LIN {X -6.617,Y -42.351,Z -210.966,A -90.000,B 90.000,C 0.000} C_DIS
LIN {X -6.280,Y -42.371,Z -210.884,A -90.000,B 90.000,C 0.000} C_DIS
LIN {X -6.014,Y -42.388,Z -210.830,A -90.000,B 90.000,C 0.000} C_DIS
LIN {X -5.294,Y -42.439,Z -210.703,A -90.000,B 90.000,C 0.000} C_DIS
LIN {X -5.055,Y -42.457,Z -210.668,A -90.000,B 90.000,C 0.000} C_DIS
LIN {X -4.913,Y -42.469,Z -210.653,A -90.000,B 90.000,C 0.000} C_DIS
LIN {X -4.678,Y -42.489,Z -210.636,A -90.000,B 90.000,C 0.000} C_DIS
LIN {X -4.349,Y -42.521,Z -210.624,A -90.000,B 90.000,C 0.000} C_DIS
LIN {X -4.051,Y -42.551,Z -210.626,A -90.000,B 90.000,C 0.000} C_DIS
LIN {X -3.773,Y -42.581,Z -210.638,A -90.000,B 90.000,C 0.000} C_DIS
LIN {X -3.082,Y -42.611,Z -210.410,A -90.000,B 90.000,C 0.000} C_DIS
LIN {X -2.709,Y -42.612,Z -210.205,A -90.000,B 90.000,C 0.000} C_DIS
LIN {X -2.509,Y -42.614,Z -210.106,A -90.000,B 90.000,C 0.000} C_DIS
LIN {X -2.183,Y -42.620,Z -209.957,A -90.000,B 90.000,C 0.000} C_DIS
LIN {X -2.016,Y -42.624,Z -209.889,A -90.000,B 90.000,C 0.000} C_DIS
LIN {X -1.766,Y -42.632,Z -209.800,A -90.000,B 90.000,C 0.000} C_DIS
LIN {X -1.327,Y -42.645,Z -209.666,A -90.000,B 90.000,C 0.000} C_DIS
LIN {X -1.055,Y -42.655,Z -209.597,A -90.000,B 90.000,C 0.000} C_DIS
LIN {X -0.921,Y -42.661,Z -209.569,A -90.000,B 90.000,C 0.000} C_DIS
LIN {X -0.790,Y -42.670,Z -209.542,A -90.000,B 90.000,C 0.000} C_DIS
LIN {X -0.184,Y -42.653,Z -208.934,A -90.000,B 90.000,C 0.000} C_DIS
LIN {X -0.036,Y -42.650,Z -208.795,A -90.000,B 90.000,C 0.000} C_DIS
LIN {X 0.358,Y -42.637,Z -208.433,A -90.000,B 90.000,C 0.000} C_DIS
LIN {X 2.070,Y -42.427,Z -205.938,A -90.000,B 90.000,C 0.000} C_DIS
LIN {X 2.234,Y -42.419,Z -205.708,A -90.000,B 90.000,C 0.000} C_DIS
LIN {X 2.733,Y -42.394,Z -205.030,A -90.000,B 90.000,C 0.000} C_DIS
LIN {X 3.270,Y -42.350,Z -204.307,A -90.000,B 90.000,C 0.000} C_DIS
LIN {X 4.497,Y -42.165,Z -202.176,A -90.000,B 90.000,C 0.000} C_DIS
LIN {X 4.596,Y -42.148,Z -202.016,A -90.000,B 90.000,C 0.000} C_DIS
LIN {X 6.267,Y -41.968,Z -199.269,A -90.000,B 90.000,C 0.000} C_DIS
LIN {X 6.453,Y -41.942,Z -198.966,A -90.000,B 90.000,C 0.000} C_DIS
LIN {X 6.699,Y -41.891,Z -198.498,A -90.000,B 90.000,C 0.000} C_DIS
LIN {X 7.020,Y -41.828,Z -197.909,A -90.000,B 90.000,C 0.000} C_DIS
LIN {X 7.766,Y -41.714,Z -196.530,A -90.000,B 90.000,C 0.000} C_DIS
LIN {X 7.949,Y -41.691,Z -196.212,A -90.000,B 90.000,C 0.000} C_DIS
LIN {X 9.284,Y -41.563,Z -193.973,A -90.000,B 90.000,C 0.000} C_DIS
LIN {X 9.444,Y -41.549,Z -193.721,A -90.000,B 90.000,C 0.000} C_DIS
LIN {X 9.586,Y -41.533,Z -193.478,A -90.000,B 90.000,C 0.000} C_DIS
LIN {X 10.446,Y -41.437,Z -192.021,A -90.000,B 90.000,C 0.000} C_DIS
LIN {X 10.972,Y -41.378,Z -191.131,A -90.000,B 90.000,C 0.000} C_DIS
LIN {X 11.489,Y -41.308,Z -190.267,A -90.000,B 90.000,C 0.000} C_DIS
LIN {X 11.489,Y -60.000,Z -190.267,A -90.000,B 90.000,C 0.000} C_DIS
LIN {X -12.262,Y -60.000,Z -210.299,A -90.000,B 90.000,C 0.000} C_DIS
LIN {X -12.262,Y -41.308,Z -210.299,A -90.000,B 90.000,C 0.000} C_DIS
LIN {X -11.900,Y -41.347,Z -210.184,A -90.000,B 90.000,C 0.000} C_DIS
LIN {X -11.506,Y -41.394,Z -210.074,A -90.000,B 90.000,C 0.000} C_DIS
LIN {X -11.190,Y -41.436,Z -210.001,A -90.000,B 90.000,C 0.000} C_DIS
LIN {X -11.051,Y -41.456,Z -209.972,A -90.000,B 90.000,C 0.000} C_DIS
LIN {X -10.725,Y -41.505,Z -209.911,A -90.000,B 90.000,C 0.000} C_DIS
LIN {X -10.408,Y -41.557,Z -209.864,A -90.000,B 90.000,C 0.000} C_DIS
LIN {X -9.634,Y -41.647,Z -209.785,A -90.000,B 90.000,C 0.000} C_DIS
LIN {X -9.462,Y -41.666,Z -209.768,A -90.000,B 90.000,C 0.000} C_DIS
LIN {X -9.236,Y -41.684,Z -209.720,A -90.000,B 90.000,C 0.000} C_DIS
LIN {X -8.688,Y -41.735,Z -209.603,A -90.000,B 90.000,C 0.000} C_DIS
LIN {X -8.324,Y -41.772,Z -209.525,A -90.000,B 90.000,C 0.000} C_DIS
LIN {X -8.206,Y -41.777,Z -209.473,A -90.000,B 90.000,C 0.000} C_DIS
LIN {X -8.132,Y -41.782,Z -209.447,A -90.000,B 90.000,C 0.000} C_DIS
LIN {X -7.916,Y -41.793,Z -209.356,A -90.000,B 90.000,C 0.000} C_DIS
LIN {X -7.715,Y -41.806,Z -209.283,A -90.000,B 90.000,C 0.000} C_DIS
LIN {X -7.389,Y -41.830,Z -209.175,A -90.000,B 90.000,C 0.000} C_DIS
LIN {X -7.217,Y -41.843,Z -209.124,A -90.000,B 90.000,C 0.000} C_DIS
LIN {X -7.050,Y -41.858,Z -209.077,A -90.000,B 90.000,C 0.000} C_DIS
LIN {X -6.640,Y -41.895,Z -208.975,A -90.000,B 90.000,C 0.000} C_DIS
LIN {X -6.321,Y -41.928,Z -208.907,A -90.000,B 90.000,C 0.000} C_DIS
LIN {X -5.544,Y -42.012,Z -208.765,A -90.000,B 90.000,C 0.000} C_DIS
LIN {X -5.228,Y -42.049,Z -208.717,A -90.000,B 90.000,C 0.000} C_DIS
LIN {X -5.016,Y -42.076,Z -208.694,A -90.000,B 90.000,C 0.000} C_DIS
LIN {X -4.805,Y -42.103,Z -208.678,A -90.000,B 90.000,C 0.000} C_DIS
LIN {X -4.663,Y -42.117,Z -208.671,A -90.000,B 90.000,C 0.000} C_DIS
LIN {X -4.355,Y -42.149,Z -208.659,A -90.000,B 90.000,C 0.000} C_DIS
LIN {X -4.025,Y -42.185,Z -208.660,A -90.000,B 90.000,C 0.000} C_DIS
LIN {X -3.857,Y -42.193,Z -208.605,A -90.000,B 90.000,C 0.000} C_DIS
LIN {X -3.580,Y -42.193,Z -208.454,A -90.000,B 90.000,C 0.000} C_DIS
LIN {X -3.315,Y -42.196,Z -208.323,A -90.000,B 90.000,C 0.000} C_DIS
LIN {X -2.989,Y -42.202,Z -208.174,A -90.000,B 90.000,C 0.000} C_DIS
LIN {X -2.844,Y -42.206,Z -208.114,A -90.000,B 90.000,C 0.000} C_DIS
LIN {X -2.716,Y -42.210,Z -208.062,A -90.000,B 90.000,C 0.000} C_DIS
LIN {X -2.412,Y -42.229,Z -207.951,A -90.000,B 90.000,C 0.000} C_DIS
LIN {X -2.184,Y -42.245,Z -207.877,A -90.000,B 90.000,C 0.000} C_DIS
LIN {X -1.891,Y -42.266,Z -207.785,A -90.000,B 90.000,C 0.000} C_DIS
LIN {X -1.797,Y -42.273,Z -207.758,A -90.000,B 90.000,C 0.000} C_DIS
LIN {X -1.778,Y -42.274,Z -207.753,A -90.000,B 90.000,C 0.000} C_DIS
LIN {X -1.529,Y -42.262,Z -207.506,A -90.000,B 90.000,C 0.000} C_DIS
LIN {X -1.146,Y -42.248,Z -207.152,A -90.000,B 90.000,C 0.000} C_DIS
LIN {X -0.566,Y -42.173,Z -206.308,A -90.000,B 90.000,C 0.000} C_DIS
LIN {X 0.472,Y -42.006,Z -204.812,A -90.000,B 90.000,C 0.000} C_DIS
LIN {X 0.654,Y -41.989,Z -204.560,A -90.000,B 90.000,C 0.000} C_DIS
LIN {X 1.498,Y -41.917,Z -203.424,A -90.000,B 90.000,C 0.000} C_DIS
LIN {X 1.621,Y -41.903,Z -203.259,A -90.000,B 90.000,C 0.000} C_DIS
LIN {X 2.825,Y -41.665,Z -201.198,A -90.000,B 90.000,C 0.000} C_DIS
LIN {X 2.924,Y -41.649,Z -201.038,A -90.000,B 90.000,C 0.000} C_DIS
LIN {X 3.144,Y -41.624,Z -200.676,A -90.000,B 90.000,C 0.000} C_DIS
LIN {X 3.568,Y -41.563,Z -199.988,A -90.000,B 90.000,C 0.000} C_DIS
LIN {X 4.759,Y -41.384,Z -198.058,A -90.000,B 90.000,C 0.000} C_DIS
LIN {X 4.988,Y -41.334,Z -197.625,A -90.000,B 90.000,C 0.000} C_DIS
LIN {X 5.113,Y -41.308,Z -197.396,A -90.000,B 90.000,C 0.000} C_DIS
LIN {X 5.113,Y -60.000,Z -197.396,A -90.000,B 90.000,C 0.000} C_DIS
LIN {X -7.484,Y -60.000,Z -207.204,A -90.000,B 90.000,C 0.000} C_DIS
LIN {X -7.484,Y -41.308,Z -207.204,A -90.000,B 90.000,C 0.000} C_DIS
LIN {X -6.986,Y -41.355,Z -207.081,A -90.000,B 90.000,C 0.000} C_DIS
LIN {X -6.613,Y -41.394,Z -207.002,A -90.000,B 90.000,C 0.000} C_DIS
LIN {X -5.770,Y -41.488,Z -206.848,A -90.000,B 90.000,C 0.000} C_DIS
LIN {X -5.453,Y -41.526,Z -206.800,A -90.000,B 90.000,C 0.000} C_DIS
LIN {X -5.161,Y -41.564,Z -206.766,A -90.000,B 90.000,C 0.000} C_DIS
LIN {X -4.857,Y -41.606,Z -206.741,A -90.000,B 90.000,C 0.000} C_DIS
LIN {X -4.638,Y -41.638,Z -206.729,A -90.000,B 90.000,C 0.000} C_DIS
LIN {X -4.424,Y -41.670,Z -206.718,A -90.000,B 90.000,C 0.000} C_DIS
LIN {X -4.164,Y -41.683,Z -206.587,A -90.000,B 90.000,C 0.000} C_DIS
LIN {X -3.727,Y -41.709,Z -206.382,A -90.000,B 90.000,C 0.000} C_DIS
LIN {X -3.429,Y -41.730,Z -206.256,A -90.000,B 90.000,C 0.000} C_DIS
LIN {X -3.096,Y -41.758,Z -206.131,A -90.000,B 90.000,C 0.000} C_DIS
LIN {X -2.982,Y -41.767,Z -206.090,A -90.000,B 90.000,C 0.000} C_DIS
LIN {X -2.792,Y -41.785,Z -206.027,A -90.000,B 90.000,C 0.000} C_DIS
LIN {X -2.642,Y -41.778,Z -205.889,A -90.000,B 90.000,C 0.000} C_DIS
LIN {X -1.365,Y -41.555,Z -204.057,A -90.000,B 90.000,C 0.000} C_DIS
LIN {X -1.115,Y -41.506,Z -203.702,A -90.000,B 90.000,C 0.000} C_DIS
LIN {X -1.083,Y -41.500,Z -203.658,A -90.000,B 90.000,C 0.000} C_DIS
LIN {X -0.913,Y -41.478,Z -203.427,A -90.000,B 90.000,C 0.000} C_DIS
LIN {X -0.012,Y -41.369,Z -202.229,A -90.000,B 90.000,C 0.000} C_DIS
LIN {X 0.278,Y -41.308,Z -201.734,A -90.000,B 90.000,C 0.000} C_DIS
LIN {X 0.278,Y -60.000,Z -201.734,A -90.000,B 90.000,C 0.000} C_DIS
LIN {X -23.050,Y -60.000,Z -133.482,A -90.000,B 90.000,C 0.000} C_DIS
LIN {X -23.050,Y -41.308,Z -133.482,A -90.000,B 90.000,C 0.000} C_DIS
LIN {X -23.070,Y -41.317,Z -133.385,A -90.000,B 90.000,C 0.000} C_DIS
LIN {X -23.094,Y -41.329,Z -133.252,A -90.000,B 90.000,C 0.000} C_DIS
LIN {X -23.314,Y -41.439,Z -131.911,A -90.000,B 90.000,C 0.000} C_DIS
LIN {X -23.329,Y -41.449,Z -131.802,A -90.000,B 90.000,C 0.000} C_DIS
LIN {X -23.404,Y -41.504,Z -131.165,A -90.000,B 90.000,C 0.000} C_DIS
LIN {X -23.458,Y -41.576,Z -130.456,A -90.000,B 90.000,C 0.000} C_DIS
LIN {X -23.470,Y -41.599,Z -130.246,A -90.000,B 90.000,C 0.000} C_DIS
LIN {X -23.473,Y -41.621,Z -130.071,A -90.000,B 90.000,C 0.000} C_DIS
LIN {X -23.473,Y -41.634,Z -129.976,A -90.000,B 90.000,C 0.000} C_DIS
LIN {X -23.470,Y -41.652,Z -129.815,A -90.000,B 90.000,C 0.000} C_DIS
LIN {X -23.462,Y -41.671,Z -129.600,A -90.000,B 90.000,C 0.000} C_DIS
LIN {X -23.484,Y -41.694,Z -129.239,A -90.000,B 90.000,C 0.000} C_DIS
LIN {X -23.533,Y -41.742,Z -128.346,A -90.000,B 90.000,C 0.000} C_DIS
LIN {X -23.555,Y -41.785,Z -127.639,A -90.000,B 90.000,C 0.000} C_DIS
LIN {X -23.575,Y -41.830,Z -127.087,A -90.000,B 90.000,C 0.000} C_DIS
LIN {X -23.574,Y -41.836,Z -127.029,A -90.000,B 90.000,C 0.000} C_DIS
LIN {X -23.576,Y -41.850,Z -126.858,A -90.000,B 90.000,C 0.000} C_DIS
LIN {X -23.569,Y -41.874,Z -126.625,A -90.000,B 90.000,C 0.000} C_DIS
LIN {X -23.533,Y -41.955,Z -125.844,A -90.000,B 90.000,C 0.000} C_DIS
LIN {X -23.511,Y -41.992,Z -125.277,A -90.000,B 90.000,C 0.000} C_DIS
LIN {X -23.515,Y -41.993,Z -125.243,A -90.000,B 90.000,C 0.000} C_DIS
LIN {X -23.643,Y -42.000,Z -124.602,A -90.000,B 90.000,C 0.000} C_DIS
LIN {X -23.792,Y -42.013,Z -123.757,A -90.000,B 90.000,C 0.000} C_DIS
LIN {X -24.070,Y -42.088,Z -122.244,A -90.000,B 90.000,C 0.000} C_DIS
LIN {X -24.088,Y -42.092,Z -122.140,A -90.000,B 90.000,C 0.000} C_DIS
LIN {X -24.107,Y -42.093,Z -122.030,A -90.000,B 90.000,C 0.000} C_DIS
LIN {X -24.170,Y -42.098,Z -121.672,A -90.000,B 90.000,C 0.000} C_DIS
LIN {X -24.188,Y -42.102,Z -121.571,A -90.000,B 90.000,C 0.000} C_DIS
LIN {X -24.313,Y -42.107,Z -121.167,A -90.000,B 90.000,C 0.000} C_DIS
LIN {X -24.362,Y -42.107,Z -121.018,A -90.000,B 90.000,C 0.000} C_DIS
LIN {X -24.809,Y -42.092,Z -119.638,A -90.000,B 90.000,C 0.000} C_DIS
LIN {X -25.186,Y -42.121,Z -118.503,A -90.000,B 90.000,C 0.000} C_DIS
LIN {X -25.572,Y -42.137,Z -117.266,A -90.000,B 90.000,C 0.000} C_DIS
LIN {X -25.886,Y -42.145,Z -116.322,A -90.000,B 90.000,C 0.000} C_DIS
LIN {X -25.961,Y -42.146,Z -116.092,A -90.000,B 90.000,C 0.000} C_DIS
LIN {X -26.400,Y -42.139,Z -114.737,A -90.000,B 90.000,C 0.000} C_DIS
LIN {X -26.782,Y -42.128,Z -113.563,A -90.000,B 90.000,C 0.000} C_DIS
LIN {X -27.447,Y -42.107,Z -111.546,A -90.000,B 90.000,C 0.000} C_DIS
LIN {X -27.639,Y -42.097,Z -110.961,A -90.000,B 90.000,C 0.000} C_DIS
LIN {X -27.709,Y -42.085,Z -110.741,A -90.000,B 90.000,C 0.000} C_DIS
LIN {X -27.755,Y -42.074,Z -110.581,A -90.000,B 90.000,C 0.000} C_DIS
LIN {X -27.902,Y -42.042,Z -110.029,A -90.000,B 90.000,C 0.000} C_DIS
LIN {X -27.980,Y -42.025,Z -109.706,A -90.000,B 90.000,C 0.000} C_DIS
LIN {X -28.117,Y -41.997,Z -109.053,A -90.000,B 90.000,C 0.000} C_DIS
LIN {X -28.358,Y -41.959,Z -107.920,A -90.000,B 90.000,C 0.000} C_DIS
LIN {X -28.564,Y -41.915,Z -106.996,A -90.000,B 90.000,C 0.000} C_DIS
LIN {X -28.601,Y -41.908,Z -106.827,A -90.000,B 90.000,C 0.000} C_DIS
LIN {X -28.724,Y -41.886,Z -106.164,A -90.000,B 90.000,C 0.000} C_DIS
LIN {X -28.845,Y -41.853,Z -105.495,A -90.000,B 90.000,C 0.000} C_DIS
LIN {X -28.878,Y -41.839,Z -105.307,A -90.000,B 90.000,C 0.000} C_DIS
LIN {X -29.130,Y -41.699,Z -103.813,A -90.000,B 90.000,C 0.000} C_DIS
LIN {X -29.182,Y -41.668,Z -103.454,A -90.000,B 90.000,C 0.000} C_DIS
LIN {X -29.224,Y -41.644,Z -103.086,A -90.000,B 90.000,C 0.000} C_DIS
LIN {X -29.270,Y -41.615,Z -102.509,A -90.000,B 90.000,C 0.000} C_DIS
LIN {X -29.284,Y -41.604,Z -102.259,A -90.000,B 90.000,C 0.000} C_DIS
LIN {X -29.288,Y -41.597,Z -101.997,A -90.000,B 90.000,C 0.000} C_DIS
LIN {X -29.280,Y -41.590,Z -101.741,A -90.000,B 90.000,C 0.000} C_DIS
LIN {X -29.250,Y -41.584,Z -101.188,A -90.000,B 90.000,C 0.000} C_DIS
LIN {X -29.178,Y -41.548,Z -100.027,A -90.000,B 90.000,C 0.000} C_DIS
LIN {X -29.153,Y -41.527,Z -99.698,A -90.000,B 90.000,C 0.000} C_DIS
LIN {X -29.138,Y -41.516,Z -99.489,A -90.000,B 90.000,C 0.000} C_DIS
LIN {X -29.120,Y -41.500,Z -99.279,A -90.000,B 90.000,C 0.000} C_DIS
LIN {X -29.077,Y -41.476,Z -98.905,A -90.000,B 90.000,C 0.000} C_DIS
LIN {X -29.047,Y -41.466,Z -98.703,A -90.000,B 90.000,C 0.000} C_DIS
LIN {X -29.015,Y -41.459,Z -98.520,A -90.000,B 90.000,C 0.000} C_DIS
LIN {X -28.923,Y -41.447,Z -98.052,A -90.000,B 90.000,C 0.000} C_DIS
LIN {X -28.723,Y -41.430,Z -96.999,A -90.000,B 90.000,C 0.000} C_DIS
LIN {X -28.657,Y -41.423,Z -96.681,A -90.000,B 90.000,C 0.000} C_DIS
LIN {X -28.528,Y -41.392,Z -96.095,A -90.000,B 90.000,C 0.000} C_DIS
LIN {X -28.491,Y -41.386,Z -95.924,A -90.000,B 90.000,C 0.000} C_DIS
LIN {X -28.434,Y -41.380,Z -95.697,A -90.000,B 90.000,C 0.000} C_DIS
LIN {X -28.370,Y -41.376,Z -95.462,A -90.000,B 90.000,C 0.000} C_DIS
LIN {X -28.232,Y -41.376,Z -95.022,A -90.000,B 90.000,C 0.000} C_DIS
LIN {X -28.161,Y -41.380,Z -94.821,A -90.000,B 90.000,C 0.000} C_DIS
LIN {X -27.995,Y -41.393,Z -94.384,A -90.000,B 90.000,C 0.000} C_DIS
LIN {X -27.971,Y -41.392,Z -94.325,A -90.000,B 90.000,C 0.000} C_DIS
LIN {X -27.835,Y -41.387,Z -93.984,A -90.000,B 90.000,C 0.000} C_DIS
LIN {X -27.746,Y -41.381,Z -93.769,A -90.000,B 90.000,C 0.000} C_DIS
LIN {X -27.107,Y -41.358,Z -92.328,A -90.000,B 90.000,C 0.000} C_DIS
LIN {X -26.960,Y -41.359,Z -92.025,A -90.000,B 90.000,C 0.000} C_DIS
LIN {X -26.939,Y -41.360,Z -91.984,A -90.000,B 90.000,C 0.000} C_DIS
LIN {X -26.749,Y -41.354,Z -91.643,A -90.000,B 90.000,C 0.000} C_DIS
LIN {X -26.597,Y -41.354,Z -91.391,A -90.000,B 90.000,C 0.000} C_DIS
LIN {X -26.044,Y -41.374,Z -90.536,A -90.000,B 90.000,C 0.000} C_DIS
LIN {X -25.785,Y -41.388,Z -90.154,A -90.000,B 90.000,C 0.000} C_DIS
LIN {X -25.678,Y -41.396,Z -89.994,A -90.000,B 90.000,C 0.000} C_DIS
LIN {X -25.507,Y -41.402,Z -89.745,A -90.000,B 90.000,C 0.000} C_DIS
LIN {X -25.112,Y -41.397,Z -89.178,A -90.000,B 90.000,C 0.000} C_DIS
LIN {X -24.983,Y -41.397,Z -89.006,A -90.000,B 90.000,C 0.000} C_DIS
LIN {X -24.826,Y -41.399,Z -88.802,A -90.000,B 90.000,C 0.000} C_DIS
LIN {X -24.722,Y -41.402,Z -88.675,A -90.000,B 90.000,C 0.000} C_DIS
LIN {X -24.486,Y -41.412,Z -88.401,A -90.000,B 90.000,C 0.000} C_DIS
LIN {X -23.946,Y -41.445,Z -87.813,A -90.000,B 90.000,C 0.000} C_DIS
LIN {X -23.608,Y -41.453,Z -87.454,A -90.000,B 90.000,C 0.000} C_DIS
LIN {X -22.465,Y -41.470,Z -86.254,A -90.000,B 90.000,C 0.000} C_DIS
LIN {X -22.294,Y -41.476,Z -86.088,A -90.000,B 90.000,C 0.000} C_DIS
LIN {X -22.148,Y -41.484,Z -85.957,A -90.000,B 90.000,C 0.000} C_DIS
LIN {X -21.990,Y -41.494,Z -85.821,A -90.000,B 90.000,C 0.000} C_DIS
LIN {X -21.611,Y -41.517,Z -85.511,A -90.000,B 90.000,C 0.000} C_DIS
LIN {X -21.025,Y -41.548,Z -85.034,A -90.000,B 90.000,C 0.000} C_DIS
LIN {X -20.092,Y -41.578,Z -84.281,A -90.000,B 90.000,C 0.000} C_DIS
LIN {X -19.821,Y -41.583,Z -84.065,A -90.000,B 90.000,C 0.000} C_DIS
LIN {X -19.531,Y -41.587,Z -83.835,A -90.000,B 90.000,C 0.000} C_DIS
LIN {X -19.253,Y -41.588,Z -83.630,A -90.000,B 90.000,C 0.000} C_DIS
LIN {X -19.000,Y -41.592,Z -83.456,A -90.000,B 90.000,C 0.000} C_DIS
LIN {X -18.820,Y -41.594,Z -83.345,A -90.000,B 90.000,C 0.000} C_DIS
LIN {X -18.604,Y -41.598,Z -83.216,A -90.000,B 90.000,C 0.000} C_DIS
LIN {X -18.307,Y -41.608,Z -83.053,A -90.000,B 90.000,C 0.000} C_DIS
LIN {X -17.615,Y -41.631,Z -82.678,A -90.000,B 90.000,C 0.000} C_DIS
LIN {X -16.357,Y -41.640,Z -82.007,A -90.000,B 90.000,C 0.000} C_DIS
LIN {X -16.157,Y -41.644,Z -81.909,A -90.000,B 90.000,C 0.000} C_DIS
LIN {X -15.796,Y -41.652,Z -81.743,A -90.000,B 90.000,C 0.000} C_DIS
LIN {X -15.527,Y -41.656,Z -81.627,A -90.000,B 90.000,C 0.000} C_DIS
LIN {X -15.356,Y -41.651,Z -81.555,A -90.000,B 90.000,C 0.000} C_DIS
LIN {X -14.632,Y -41.625,Z -81.254,A -90.000,B 90.000,C 0.000} C_DIS
LIN {X -14.380,Y -41.619,Z -81.159,A -90.000,B 90.000,C 0.000} C_DIS
LIN {X -14.313,Y -41.617,Z -81.134,A -90.000,B 90.000,C 0.000} C_DIS
LIN {X -13.263,Y -41.602,Z -80.775,A -90.000,B 90.000,C 0.000} C_DIS
LIN {X -13.022,Y -41.593,Z -80.697,A -90.000,B 90.000,C 0.000} C_DIS
LIN {X -12.835,Y -41.588,Z -80.644,A -90.000,B 90.000,C 0.000} C_DIS
LIN {X -12.618,Y -41.584,Z -80.588,A -90.000,B 90.000,C 0.000} C_DIS
LIN {X -11.074,Y -41.571,Z -80.238,A -90.000,B 90.000,C 0.000} C_DIS
LIN {X -10.804,Y -41.562,Z -80.179,A -90.000,B 90.000,C 0.000} C_DIS
LIN {X -9.749,Y -41.484,Z -79.972,A -90.000,B 90.000,C 0.000} C_DIS
LIN {X -9.567,Y -41.473,Z -79.943,A -90.000,B 90.000,C 0.000} C_DIS
LIN {X -9.291,Y -41.458,Z -79.904,A -90.000,B 90.000,C 0.000} C_DIS
LIN {X -8.345,Y -41.422,Z -79.809,A -90.000,B 90.000,C 0.000} C_DIS
LIN {X -8.092,Y -41.407,Z -79.786,A -90.000,B 90.000,C 0.000} C_DIS
LIN {X -6.966,Y -41.348,Z -79.697,A -90.000,B 90.000,C 0.000} C_DIS
LIN {X -6.019,Y -41.308,Z -79.651,A -90.000,B 90.000,C 0.000} C_DIS
LIN {X -6.019,Y -60.000,Z -79.651,A -90.000,B 90.000,C 0.000} C_DIS
LIN {X 25.151,Y -60.000,Z -82.979,A -90.000,B 90.000,C 0.000} C_DIS
LIN {X 25.151,Y -41.308,Z -82.979,A -90.000,B 90.000,C 0.000} C_DIS
LIN {X 25.401,Y -41.345,Z -82.958,A -90.000,B 90.000,C 0.000} C_DIS
LIN {X 26.505,Y -41.507,Z -82.878,A -90.000,B 90.000,C 0.000} C_DIS
LIN {X 27.673,Y -41.657,Z -82.800,A -90.000,B 90.000,C 0.000} C_DIS
LIN {X 27.698,Y -41.660,Z -82.799,A -90.000,B 90.000,C 0.000} C_DIS
LIN {X 28.017,Y -41.696,Z -82.752,A -90.000,B 90.000,C 0.000} C_DIS
LIN {X 28.158,Y -41.713,Z -82.736,A -90.000,B 90.000,C 0.000} C_DIS
LIN {X 28.252,Y -41.725,Z -82.727,A -90.000,B 90.000,C 0.000} C_DIS
LIN {X 28.530,Y -41.760,Z -82.709,A -90.000,B 90.000,C 0.000} C_DIS
LIN {X 29.119,Y -41.837,Z -82.692,A -90.000,B 90.000,C 0.000} C_DIS
LIN {X 29.519,Y -41.890,Z -82.684,A -90.000,B 90.000,C 0.000} C_DIS
LIN {X 29.940,Y -41.940,Z -82.676,A -90.000,B 90.000,C 0.000} C_DIS
LIN {X 31.269,Y -42.060,Z -82.659,A -90.000,B 90.000,C 0.000} C_DIS
LIN {X 32.112,Y -42.118,Z -82.572,A -90.000,B 90.000,C 0.000} C_DIS
LIN {X 32.318,Y -42.133,Z -82.559,A -90.000,B 90.000,C 0.000} C_DIS
LIN {X 32.590,Y -42.153,Z -82.550,A -90.000,B 90.000,C 0.000} C_DIS
LIN {X 32.942,Y -42.181,Z -82.546,A -90.000,B 90.000,C 0.000} C_DIS
LIN {X 33.071,Y -42.192,Z -82.549,A -90.000,B 90.000,C 0.000} C_DIS
LIN {X 33.237,Y -42.204,Z -82.556,A -90.000,B 90.000,C 0.000} C_DIS
LIN {X 33.498,Y -42.212,Z -82.568,A -90.000,B 90.000,C 0.000} C_DIS
LIN {X 33.767,Y -42.216,Z -82.581,A -90.000,B 90.000,C 0.000} C_DIS
LIN {X 34.438,Y -42.216,Z -82.618,A -90.000,B 90.000,C 0.000} C_DIS
LIN {X 34.735,Y -42.217,Z -82.645,A -90.000,B 90.000,C 0.000} C_DIS
LIN {X 34.872,Y -42.218,Z -82.662,A -90.000,B 90.000,C 0.000} C_DIS
LIN {X 35.054,Y -42.220,Z -82.691,A -90.000,B 90.000,C 0.000} C_DIS
LIN {X 35.259,Y -42.222,Z -82.728,A -90.000,B 90.000,C 0.000} C_DIS
LIN {X 35.802,Y -42.227,Z -82.837,A -90.000,B 90.000,C 0.000} C_DIS
LIN {X 36.714,Y -42.242,Z -83.021,A -90.000,B 90.000,C 0.000} C_DIS
LIN {X 37.139,Y -42.247,Z -83.108,A -90.000,B 90.000,C 0.000} C_DIS
LIN {X 37.332,Y -42.247,Z -83.134,A -90.000,B 90.000,C 0.000} C_DIS
LIN {X 37.517,Y -42.248,Z -83.166,A -90.000,B 90.000,C 0.000} C_DIS
LIN {X 37.642,Y -42.246,Z -83.190,A -90.000,B 90.000,C 0.000} C_DIS
LIN {X 37.947,Y -42.234,Z -83.255,A -90.000,B 90.000,C 0.000} C_DIS
LIN {X 38.137,Y -42.228,Z -83.303,A -90.000,B 90.000,C 0.000} C_DIS
LIN {X 38.362,Y -42.221,Z -83.362,A -90.000,B 90.000,C 0.000} C_DIS
LIN {X 38.756,Y -42.210,Z -83.482,A -90.000,B 90.000,C 0.000} C_DIS
LIN {X 39.315,Y -42.195,Z -83.661,A -90.000,B 90.000,C 0.000} C_DIS
LIN {X 40.217,Y -42.193,Z -83.945,A -90.000,B 90.000,C 0.000} C_DIS
LIN {X 40.592,Y -42.178,Z -84.068,A -90.000,B 90.000,C 0.000} C_DIS
LIN {X 40.724,Y -42.173,Z -84.115,A -90.000,B 90.000,C 0.000} C_DIS
LIN {X 40.993,Y -42.165,Z -84.219,A -90.000,B 90.000,C 0.000} C_DIS
LIN {X 41.178,Y -42.160,Z -84.299,A -90.000,B 90.000,C 0.000} C_DIS
LIN {X 41.409,Y -42.154,Z -84.403,A -90.000,B 90.000,C 0.000} C_DIS
LIN {X 41.680,Y -42.148,Z -84.532,A -90.000,B 90.000,C 0.000} C_DIS
LIN {X 41.769,Y -42.150,Z -84.573,A -90.000,B 90.000,C 0.000} C_DIS
LIN {X 42.730,Y -42.131,Z -85.032,A -90.000,B 90.000,C 0.000} C_DIS
LIN {X 43.145,Y -42.123,Z -85.233,A -90.000,B 90.000,C 0.000} C_DIS
LIN {X 43.266,Y -42.121,Z -85.296,A -90.000,B 90.000,C 0.000} C_DIS
LIN {X 43.406,Y -42.119,Z -85.373,A -90.000,B 90.000,C 0.000} C_DIS
LIN {X 43.868,Y -42.093,Z -85.640,A -90.000,B 90.000,C 0.000} C_DIS
LIN {X 44.070,Y -42.083,Z -85.767,A -90.000,B 90.000,C 0.000} C_DIS
LIN {X 44.306,Y -42.072,Z -85.930,A -90.000,B 90.000,C 0.000} C_DIS
LIN {X 44.337,Y -42.071,Z -85.953,A -90.000,B 90.000,C 0.000} C_DIS
LIN {X 44.520,Y -42.075,Z -86.085,A -90.000,B 90.000,C 0.000} C_DIS
LIN {X 44.824,Y -42.070,Z -86.257,A -90.000,B 90.000,C 0.000} C_DIS
LIN {X 45.576,Y -42.041,Z -86.685,A -90.000,B 90.000,C 0.000} C_DIS
LIN {X 45.736,Y -42.033,Z -86.781,A -90.000,B 90.000,C 0.000} C_DIS
LIN {X 45.953,Y -42.024,Z -86.921,A -90.000,B 90.000,C 0.000} C_DIS
LIN {X 46.138,Y -42.017,Z -87.050,A -90.000,B 90.000,C 0.000} C_DIS
LIN {X 46.527,Y -42.004,Z -87.334,A -90.000,B 90.000,C 0.000} C_DIS
LIN {X 46.855,Y -41.986,Z -87.580,A -90.000,B 90.000,C 0.000} C_DIS
LIN {X 47.338,Y -41.957,Z -87.944,A -90.000,B 90.000,C 0.000} C_DIS
LIN {X 47.485,Y -41.948,Z -88.062,A -90.000,B 90.000,C 0.000} C_DIS
LIN {X 47.657,Y -41.947,Z -88.202,A -90.000,B 90.000,C 0.000} C_DIS
LIN {X 48.084,Y -41.944,Z -88.559,A -90.000,B 90.000,C 0.000} C_DIS
LIN {X 48.477,Y -41.930,Z -88.894,A -90.000,B 90.000,C 0.000} C_DIS
LIN {X 48.677,Y -41.925,Z -89.081,A -90.000,B 90.000,C 0.000} C_DIS
LIN {X 48.825,Y -41.922,Z -89.229,A -90.000,B 90.000,C 0.000} C_DIS
LIN {X 48.926,Y -41.920,Z -89.337,A -90.000,B 90.000,C 0.000} C_DIS
LIN {X 49.697,Y -41.908,Z -90.192,A -90.000,B 90.000,C 0.000} C_DIS
LIN {X 49.759,Y -41.905,Z -90.262,A -90.000,B 90.000,C 0.000} C_DIS
LIN {X 50.273,Y -41.870,Z -90.773,A -90.000,B 90.000,C 0.000} C_DIS
LIN {X 50.447,Y -41.859,Z -90.959,A -90.000,B 90.000,C 0.000} C_DIS
LIN {X 50.646,Y -41.848,Z -91.184,A -90.000,B 90.000,C 0.000} C_DIS
LIN {X 50.826,Y -41.840,Z -91.399,A -90.000,B 90.000,C 0.000} C_DIS
LIN {X 51.215,Y -41.827,Z -91.893,A -90.000,B 90.000,C 0.000} C_DIS
LIN {X 51.328,Y -41.822,Z -92.045,A -90.000,B 90.000,C 0.000} C_DIS
LIN {X 51.423,Y -41.815,Z -92.183,A -90.000,B 90.000,C 0.000} C_DIS
LIN {X 51.554,Y -41.807,Z -92.378,A -90.000,B 90.000,C 0.000} C_DIS
LIN {X 51.611,Y -41.804,Z -92.468,A -90.000,B 90.000,C 0.000} C_DIS
LIN {X 51.718,Y -41.799,Z -92.646,A -90.000,B 90.000,C 0.000} C_DIS
LIN {X 52.404,Y -41.777,Z -93.855,A -90.000,B 90.000,C 0.000} C_DIS
LIN {X 53.286,Y -41.749,Z -95.416,A -90.000,B 90.000,C 0.000} C_DIS
LIN {X 53.574,Y -41.715,Z -95.938,A -90.000,B 90.000,C 0.000} C_DIS
LIN {X 53.677,Y -41.703,Z -96.139,A -90.000,B 90.000,C 0.000} C_DIS
LIN {X 53.802,Y -41.690,Z -96.402,A -90.000,B 90.000,C 0.000} C_DIS
LIN {X 53.855,Y -41.685,Z -96.522,A -90.000,B 90.000,C 0.000} C_DIS
LIN {X 54.017,Y -41.673,Z -96.909,A -90.000,B 90.000,C 0.000} C_DIS
LIN {X 54.194,Y -41.645,Z -97.340,A -90.000,B 90.000,C 0.000} C_DIS
LIN {X 54.288,Y -41.632,Z -97.596,A -90.000,B 90.000,C 0.000} C_DIS
LIN {X 54.326,Y -41.627,Z -97.703,A -90.000,B 90.000,C 0.000} C_DIS
LIN {X 54.551,Y -41.598,Z -98.399,A -90.000,B 90.000,C 0.000} C_DIS
LIN {X 54.643,Y -41.588,Z -98.722,A -90.000,B 90.000,C 0.000} C_DIS
LIN {X 54.747,Y -41.578,Z -99.122,A -90.000,B 90.000,C 0.000} C_DIS
LIN {X 54.843,Y -41.571,Z -99.532,A -90.000,B 90.000,C 0.000} C_DIS
LIN {X 55.081,Y -41.529,Z -100.575,A -90.000,B 90.000,C 0.000} C_DIS
LIN {X 55.243,Y -41.485,Z -101.309,A -90.000,B 90.000,C 0.000} C_DIS
LIN {X 55.273,Y -41.474,Z -101.451,A -90.000,B 90.000,C 0.000} C_DIS
LIN {X 55.318,Y -41.453,Z -101.663,A -90.000,B 90.000,C 0.000} C_DIS
LIN {X 55.355,Y -41.434,Z -101.871,A -90.000,B 90.000,C 0.000} C_DIS
LIN {X 55.403,Y -41.408,Z -102.211,A -90.000,B 90.000,C 0.000} C_DIS
LIN {X 55.428,Y -41.394,Z -102.428,A -90.000,B 90.000,C 0.000} C_DIS
LIN {X 55.540,Y -41.308,Z -104.020,A -90.000,B 90.000,C 0.000} C_DIS
LIN {X 55.540,Y -60.000,Z -104.020,A -90.000,B 90.000,C 0.000} C_DIS
LIN {X 47.858,Y -60.000,Z -81.598,A -90.000,B 90.000,C 0.000} C_DIS
LIN {X 47.858,Y -41.308,Z -81.598,A -90.000,B 90.000,C 0.000} C_DIS
LIN {X 47.690,Y -41.324,Z -81.608,A -90.000,B 90.000,C 0.000} C_DIS
LIN {X 47.343,Y -41.356,Z -81.614,A -90.000,B 90.000,C 0.000} C_DIS
LIN {X 46.537,Y -41.428,Z -81.604,A -90.000,B 90.000,C 0.000} C_DIS
LIN {X 46.220,Y -41.462,Z -81.598,A -90.000,B 90.000,C 0.000} C_DIS
LIN {X 45.787,Y -41.504,Z -81.585,A -90.000,B 90.000,C 0.000} C_DIS
LIN {X 45.664,Y -41.514,Z -81.582,A -90.000,B 90.000,C 0.000} C_DIS
LIN {X 45.515,Y -41.525,Z -81.571,A -90.000,B 90.000,C 0.000} C_DIS
LIN {X 45.297,Y -41.541,Z -81.562,A -90.000,B 90.000,C 0.000} C_DIS
LIN {X 44.674,Y -41.595,Z -81.512,A -90.000,B 90.000,C 0.000} C_DIS
LIN {X 44.318,Y -41.625,Z -81.471,A -90.000,B 90.000,C 0.000} C_DIS
LIN {X 43.773,Y -41.676,Z -81.383,A -90.000,B 90.000,C 0.000} C_DIS
LIN {X 43.571,Y -41.695,Z -81.342,A -90.000,B 90.000,C 0.000} C_DIS
LIN {X 43.194,Y -41.730,Z -81.251,A -90.000,B 90.000,C 0.000} C_DIS
LIN {X 42.955,Y -41.751,Z -81.182,A -90.000,B 90.000,C 0.000} C_DIS
LIN {X 42.754,Y -41.766,Z -81.124,A -90.000,B 90.000,C 0.000} C_DIS
LIN {X 42.111,Y -41.805,Z -80.932,A -90.000,B 90.000,C 0.000} C_DIS
LIN {X 41.675,Y -41.846,Z -81.049,A -90.000,B 90.000,C 0.000} C_DIS
LIN {X 41.410,Y -41.870,Z -81.110,A -90.000,B 90.000,C 0.000} C_DIS
LIN {X 41.035,Y -41.900,Z -81.207,A -90.000,B 90.000,C 0.000} C_DIS
LIN {X 40.892,Y -41.911,Z -81.241,A -90.000,B 90.000,C 0.000} C_DIS
LIN {X 40.338,Y -41.947,Z -81.354,A -90.000,B 90.000,C 0.000} C_DIS
LIN {X 39.958,Y -41.971,Z -81.424,A -90.000,B 90.000,C 0.000} C_DIS
LIN {X 39.368,Y -42.009,Z -81.520,A -90.000,B 90.000,C 0.000} C_DIS
LIN {X 39.219,Y -42.018,Z -81.542,A -90.000,B 90.000,C 0.000} C_DIS
LIN {X 39.804,Y -41.992,Z -81.729,A -90.000,B 90.000,C 0.000} C_DIS
LIN {X 40.431,Y -41.977,Z -81.928,A -90.000,B 90.000,C 0.000} C_DIS
LIN {X 40.828,Y -41.960,Z -82.055,A -90.000,B 90.000,C 0.000} C_DIS
LIN {X 41.240,Y -41.944,Z -82.191,A -90.000,B 90.000,C 0.000} C_DIS
LIN {X 41.437,Y -41.936,Z -82.261,A -90.000,B 90.000,C 0.000} C_DIS
LIN {X 41.776,Y -41.924,Z -82.394,A -90.000,B 90.000,C 0.000} C_DIS
LIN {X 42.028,Y -41.915,Z -82.505,A -90.000,B 90.000,C 0.000} C_DIS
LIN {X 42.291,Y -41.900,Z -82.625,A -90.000,B 90.000,C 0.000} C_DIS
LIN {X 42.496,Y -41.890,Z -82.724,A -90.000,B 90.000,C 0.000} C_DIS
LIN {X 43.692,Y -41.856,Z -83.297,A -90.000,B 90.000,C 0.000} C_DIS
LIN {X 43.866,Y -41.846,Z -83.382,A -90.000,B 90.000,C 0.000} C_DIS
LIN {X 44.061,Y -41.831,Z -83.479,A -90.000,B 90.000,C 0.000} C_DIS
LIN {X 44.252,Y -41.817,Z -83.582,A -90.000,B 90.000,C 0.000} C_DIS
LIN {X 44.628,Y -41.790,Z -83.798,A -90.000,B 90.000,C 0.000} C_DIS
LIN {X 44.910,Y -41.788,Z -83.960,A -90.000,B 90.000,C 0.000} C_DIS
LIN {X 45.152,Y -41.787,Z -84.111,A -90.000,B 90.000,C 0.000} C_DIS
LIN {X 45.185,Y -41.785,Z -84.133,A -90.000,B 90.000,C 0.000} C_DIS
LIN {X 45.470,Y -41.773,Z -84.331,A -90.000,B 90.000,C 0.000} C_DIS
LIN {X 45.597,Y -41.768,Z -84.423,A -90.000,B 90.000,C 0.000} C_DIS
LIN {X 46.395,Y -41.721,Z -84.881,A -90.000,B 90.000,C 0.000} C_DIS
LIN {X 46.653,Y -41.705,Z -85.031,A -90.000,B 90.000,C 0.000} C_DIS
LIN {X 46.867,Y -41.693,Z -85.165,A -90.000,B 90.000,C 0.000} C_DIS
LIN {X 47.068,Y -41.674,Z -85.298,A -90.000,B 90.000,C 0.000} C_DIS
LIN {X 47.321,Y -41.652,Z -85.478,A -90.000,B 90.000,C 0.000} C_DIS
LIN {X 47.493,Y -41.637,Z -85.606,A -90.000,B 90.000,C 0.000} C_DIS
LIN {X 47.864,Y -41.625,Z -85.880,A -90.000,B 90.000,C 0.000} C_DIS
LIN {X 48.284,Y -41.611,Z -86.194,A -90.000,B 90.000,C 0.000} C_DIS
LIN {X 48.557,Y -41.596,Z -86.401,A -90.000,B 90.000,C 0.000} C_DIS
LIN {X 48.811,Y -41.582,Z -86.607,A -90.000,B 90.000,C 0.000} C_DIS
LIN {X 49.265,Y -41.559,Z -86.989,A -90.000,B 90.000,C 0.000} C_DIS
LIN {X 49.780,Y -41.530,Z -87.431,A -90.000,B 90.000,C 0.000} C_DIS
LIN {X 49.974,Y -41.519,Z -87.614,A -90.000,B 90.000,C 0.000} C_DIS
LIN {X 50.079,Y -41.511,Z -87.715,A -90.000,B 90.000,C 0.000} C_DIS
LIN {X 50.275,Y -41.498,Z -87.918,A -90.000,B 90.000,C 0.000} C_DIS
LIN {X 50.406,Y -41.489,Z -88.062,A -90.000,B 90.000,C 0.000} C_DIS
LIN {X 50.606,Y -41.478,Z -88.287,A -90.000,B 90.000,C 0.000} C_DIS
LIN {X 51.166,Y -41.470,Z -88.908,A -90.000,B 90.000,C 0.000} C_DIS
LIN {X 51.354,Y -41.463,Z -89.093,A -90.000,B 90.000,C 0.000} C_DIS
LIN {X 51.688,Y -41.440,Z -89.427,A -90.000,B 90.000,C 0.000} C_DIS
LIN {X 51.936,Y -41.426,Z -89.695,A -90.000,B 90.000,C 0.000} C_DIS
LIN {X 52.136,Y -41.416,Z -89.922,A -90.000,B 90.000,C 0.000} C_DIS
LIN {X 52.367,Y -41.406,Z -90.200,A -90.000,B 90.000,C 0.000} C_DIS
LIN {X 52.774,Y -41.392,Z -90.719,A -90.000,B 90.000,C 0.000} C_DIS
LIN {X 52.938,Y -41.386,Z -90.941,A -90.000,B 90.000,C 0.000} C_DIS
LIN {X 53.079,Y -41.376,Z -91.147,A -90.000,B 90.000,C 0.000} C_DIS
LIN {X 53.225,Y -41.367,Z -91.369,A -90.000,B 90.000,C 0.000} C_DIS
LIN {X 53.385,Y -41.359,Z -91.632,A -90.000,B 90.000,C 0.000} C_DIS
LIN {X 54.099,Y -41.329,Z -92.894,A -90.000,B 90.000,C 0.000} C_DIS
LIN {X 54.322,Y -41.308,Z -93.294,A -90.000,B 90.000,C 0.000} C_DIS
LIN {X 54.322,Y -60.000,Z -93.294,A -90.000,B 90.000,C 0.000} C_DIS
LIN {X 48.608,Y -60.000,Z -83.453,A -90.000,B 90.000,C 0.000} C_DIS
LIN {X 48.608,Y -41.308,Z -83.453,A -90.000,B 90.000,C 0.000} C_DIS
LIN {X 48.591,Y -41.311,Z -83.459,A -90.000,B 90.000,C 0.000} C_DIS
LIN {X 48.053,Y -41.388,Z -83.578,A -90.000,B 90.000,C 0.000} C_DIS
LIN {X 48.217,Y -41.379,Z -83.688,A -90.000,B 90.000,C 0.000} C_DIS
LIN {X 48.486,Y -41.366,Z -83.878,A -90.000,B 90.000,C 0.000} C_DIS
LIN {X 48.542,Y -41.364,Z -83.919,A -90.000,B 90.000,C 0.000} C_DIS
LIN {X 49.183,Y -41.308,Z -84.399,A -90.000,B 90.000,C 0.000} C_DIS
LIN {X 49.183,Y -60.000,Z -84.399,A -90.000,B 90.000,C 0.000} C_DIS
LIN {X 27.831,Y -60.000,Z -80.799,A -90.000,B 90.000,C 0.000} C_DIS
LIN {X 27.831,Y -41.308,Z -80.799,A -90.000,B 90.000,C 0.000} C_DIS
LIN {X 28.069,Y -41.337,Z -80.773,A -90.000,B 90.000,C 0.000} C_DIS
LIN {X 28.181,Y -41.351,Z -80.764,A -90.000,B 90.000,C 0.000} C_DIS
LIN {X 28.521,Y -41.394,Z -80.743,A -90.000,B 90.000,C 0.000} C_DIS
LIN {X 29.324,Y -41.503,Z -80.721,A -90.000,B 90.000,C 0.000} C_DIS
LIN {X 29.947,Y -41.588,Z -80.708,A -90.000,B 90.000,C 0.000} C_DIS
LIN {X 30.287,Y -41.627,Z -80.702,A -90.000,B 90.000,C 0.000} C_DIS
LIN {X 31.182,Y -41.722,Z -80.688,A -90.000,B 90.000,C 0.000} C_DIS
LIN {X 31.968,Y -41.792,Z -80.604,A -90.000,B 90.000,C 0.000} C_DIS
LIN {X 32.274,Y -41.820,Z -80.584,A -90.000,B 90.000,C 0.000} C_DIS
LIN {X 32.594,Y -41.850,Z -80.573,A -90.000,B 90.000,C 0.000} C_DIS
LIN {X 32.901,Y -41.876,Z -80.570,A -90.000,B 90.000,C 0.000} C_DIS
LIN {X 33.012,Y -41.881,Z -80.570,A -90.000,B 90.000,C 0.000} C_DIS
LIN {X 33.303,Y -41.895,Z -80.581,A -90.000,B 90.000,C 0.000} C_DIS
LIN {X 33.639,Y -41.913,Z -80.595,A -90.000,B 90.000,C 0.000} C_DIS
LIN {X 33.540,Y -41.894,Z -80.511,A -90.000,B 90.000,C 0.000} C_DIS
LIN {X 33.452,Y -41.875,Z -80.430,A -90.000,B 90.000,C 0.000} C_DIS
LIN {X 33.352,Y -41.852,Z -80.330,A -90.000,B 90.000,C 0.000} C_DIS
LIN {X 33.226,Y -41.822,Z -80.197,A -90.000,B 90.000,C 0.000} C_DIS
LIN {X 33.198,Y -41.814,Z -80.164,A -90.000,B 90.000,C 0.000} C_DIS
LIN {X 33.105,Y -41.776,Z -80.058,A -90.000,B 90.000,C 0.000} C_DIS
LIN {X 33.045,Y -41.750,Z -79.983,A -90.000,B 90.000,C 0.000} C_DIS
LIN {X 32.939,Y -41.700,Z -79.842,A -90.000,B 90.000,C 0.000} C_DIS
LIN {X 32.881,Y -41.670,Z -79.757,A -90.000,B 90.000,C 0.000} C_DIS
LIN {X 32.771,Y -41.594,Z -79.587,A -90.000,B 90.000,C 0.000} C_DIS
LIN {X 32.715,Y -41.552,Z -79.489,A -90.000,B 90.000,C 0.000} C_DIS
LIN {X 32.633,Y -41.484,Z -79.331,A -90.000,B 90.000,C 0.000} C_DIS
LIN {X 32.581,Y -41.438,Z -79.223,A -90.000,B 90.000,C 0.000} C_DIS
LIN {X 32.545,Y -41.403,Z -79.137,A -90.000,B 90.000,C 0.000} C_DIS
LIN {X 32.498,Y -41.352,Z -79.023,A -90.000,B 90.000,C 0.000} C_DIS
LIN {X 32.462,Y -41.308,Z -78.922,A -90.000,B 90.000,C 0.000} C_DIS
LIN {X 32.462,Y -60.000,Z -78.922,A -90.000,B 90.000,C 0.000} C_DIS
LIN {X 84.746,Y -60.000,Z -104.703,A -90.000,B 90.000,C 0.000} C_DIS
LIN {X 84.746,Y -41.308,Z -104.703,A -90.000,B 90.000,C 0.000} C_DIS
LIN {X 84.701,Y -41.332,Z -104.738,A -90.000,B 90.000,C 0.000} C_DIS
LIN {X 84.534,Y -41.407,Z -104.855,A -90.000,B 90.000,C 0.000} C_DIS
LIN {X 84.256,Y -41.531,Z -105.032,A -90.000,B 90.000,C 0.000} C_DIS
LIN {X 84.165,Y -41.572,Z -105.089,A -90.000,B 90.000,C 0.000} C_DIS
LIN {X 83.833,Y -41.717,Z -105.280,A -90.000,B 90.000,C 0.000} C_DIS
LIN {X 83.694,Y -41.777,Z -105.356,A -90.000,B 90.000,C 0.000} C_DIS
LIN {X 83.593,Y -41.820,Z -105.407,A -90.000,B 90.000,C 0.000} C_DIS
LIN {X 83.434,Y -41.871,Z -105.483,A -90.000,B 90.000,C 0.000} C_DIS
LIN {X 83.150,Y -41.960,Z -105.606,A -90.000,B 90.000,C 0.000} C_DIS
LIN {X 82.889,Y -42.035,Z -105.708,A -90.000,B 90.000,C 0.000} C_DIS
LIN {X 82.625,Y -42.109,Z -105.798,A -90.000,B 90.000,C 0.000} C_DIS
LIN {X 82.300,Y -42.195,Z -105.897,A -90.000,B 90.000,C 0.000} C_DIS
LIN {X 82.099,Y -42.249,Z -105.980,A -90.000,B 90.000,C 0.000} C_DIS
LIN {X 81.805,Y -42.317,Z -106.099,A -90.000,B 90.000,C 0.000} C_DIS
LIN {X 81.037,Y -42.480,Z -106.402,A -90.000,B 90.000,C 0.000} C_DIS
LIN {X 80.916,Y -42.506,Z -106.447,A -90.000,B 90.000,C 0.000} C_DIS
LIN {X 80.629,Y -42.567,Z -106.559,A -90.000,B 90.000,C 0.000} C_DIS
LIN {X 80.329,Y -42.619,Z -106.661,A -90.000,B 90.000,C 0.000} C_DIS
LIN {X 80.141,Y -42.651,Z -106.720,A -90.000,B 90.000,C 0.000} C_DIS
LIN {X 80.082,Y -42.662,Z -106.737,A -90.000,B 90.000,C 0.000} C_DIS
LIN {X 79.854,Y -42.684,Z -106.797,A -90.000,B 90.000,C 0.000} C_DIS
LIN {X 79.559,Y -42.713,Z -106.862,A -90.000,B 90.000,C 0.000} C_DIS
LIN {X 79.363,Y -42.732,Z -106.903,A -90.000,B 90.000,C 0.000} C_DIS
LIN {X 78.983,Y -42.770,Z -106.967,A -90.000,B 90.000,C 0.000} C_DIS
LIN {X 78.787,Y -42.789,Z -106.993,A -90.000,B 90.000,C 0.000} C_DIS
LIN {X 78.501,Y -42.818,Z -107.025,A -90.000,B 90.000,C 0.000} C_DIS
LIN {X 78.279,Y -42.840,Z -107.041,A -90.000,B 90.000,C 0.000} C_DIS
LIN {X 78.023,Y -42.864,Z -107.052,A -90.000,B 90.000,C 0.000} C_DIS
LIN {X 77.794,Y -42.887,Z -107.057,A -90.000,B 90.000,C 0.000} C_DIS
LIN {X 77.690,Y -42.897,Z -107.057,A -90.000,B 90.000,C 0.000} C_DIS
LIN {X 77.347,Y -42.928,Z -107.045,A -90.000,B 90.000,C 0.000} C_DIS
LIN {X 77.071,Y -42.946,Z -107.026,A -90.000,B 90.000,C 0.000} C_DIS
LIN {X 76.821,Y -42.960,Z -107.001,A -90.000,B 90.000,C 0.000} C_DIS
LIN {X 76.647,Y -42.959,Z -106.980,A -90.000,B 90.000,C 0.000} C_DIS
LIN {X 76.468,Y -42.956,Z -106.957,A -90.000,B 90.000,C 0.000} C_DIS
LIN {X 76.245,Y -42.952,Z -106.920,A -90.000,B 90.000,C 0.000} C_DIS
LIN {X 75.996,Y -42.949,Z -106.873,A -90.000,B 90.000,C 0.000} C_DIS
LIN {X 75.737,Y -42.946,Z -106.816,A -90.000,B 90.000,C 0.000} C_DIS
LIN {X 75.558,Y -42.944,Z -106.770,A -90.000,B 90.000,C 0.000} C_DIS
LIN {X 75.257,Y -42.941,Z -106.683,A -90.000,B 90.000,C 0.000} C_DIS
LIN {X 75.082,Y -42.940,Z -106.627,A -90.000,B 90.000,C 0.000} C_DIS
LIN {X 74.620,Y -42.937,Z -106.473,A -90.000,B 90.000,C 0.000} C_DIS
LIN {X 74.393,Y -42.934,Z -106.404,A -90.000,B 90.000,C 0.000} C_DIS
LIN {X 74.320,Y -42.931,Z -106.382,A -90.000,B 90.000,C 0.000} C_DIS
LIN {X 73.862,Y -42.893,Z -106.242,A -90.000,B 90.000,C 0.000} C_DIS
LIN {X 73.756,Y -42.876,Z -106.208,A -90.000,B 90.000,C 0.000} C_DIS
LIN {X 73.470,Y -42.831,Z -106.110,A -90.000,B 90.000,C 0.000} C_DIS
LIN {X 73.156,Y -42.783,Z -105.994,A -90.000,B 90.000,C 0.000} C_DIS
LIN {X 72.968,Y -42.754,Z -105.917,A -90.000,B 90.000,C 0.000} C_DIS
LIN {X 72.570,Y -42.692,Z -105.738,A -90.000,B 90.000,C 0.000} C_DIS
LIN {X 72.444,Y -42.673,Z -105.677,A -90.000,B 90.000,C 0.000} C_DIS
LIN {X 72.233,Y -42.640,Z -105.569,A -90.000,B 90.000,C 0.000} C_DIS
LIN {X 72.090,Y -42.617,Z -105.490,A -90.000,B 90.000,C 0.000} C_DIS
LIN {X 71.905,Y -42.579,Z -105.382,A -90.000,B 90.000,C 0.000} C_DIS
LIN {X 71.682,Y -42.533,Z -105.241,A -90.000,B 90.000,C 0.000} C_DIS
LIN {X 71.591,Y -42.505,Z -105.181,A -90.000,B 90.000,C 0.000} C_DIS
LIN {X 71.535,Y -42.486,Z -105.142,A -90.000,B 90.000,C 0.000} C_DIS
LIN {X 71.405,Y -42.445,Z -105.047,A -90.000,B 90.000,C 0.000} C_DIS
LIN {X 71.144,Y -42.364,Z -104.850,A -90.000,B 90.000,C 0.000} C_DIS
LIN {X 70.943,Y -42.300,Z -104.684,A -90.000,B 90.000,C 0.000} C_DIS
LIN {X 70.719,Y -42.228,Z -104.491,A -90.000,B 90.000,C 0.000} C_DIS
LIN {X 70.477,Y -42.149,Z -104.262,A -90.000,B 90.000,C 0.000} C_DIS
LIN {X 70.362,Y -42.119,Z -104.151,A -90.000,B 90.000,C 0.000} C_DIS
LIN {X 70.274,Y -42.088,Z -104.062,A -90.000,B 90.000,C 0.000} C_DIS
LIN {X 70.130,Y -42.036,Z -103.908,A -90.000,B 90.000,C 0.000} C_DIS
LIN {X 70.012,Y -41.991,Z -103.772,A -90.000,B 90.000,C 0.000} C_DIS
LIN {X 69.887,Y -41.936,Z -103.620,A -90.000,B 90.000,C 0.000} C_DIS
LIN {X 69.721,Y -41.861,Z -103.403,A -90.000,B 90.000,C 0.000} C_DIS
LIN {X 69.547,Y -41.781,Z -103.161,A -90.000,B 90.000,C 0.000} C_DIS
LIN {X 69.507,Y -41.762,Z -103.100,A -90.000,B 90.000,C 0.000} C_DIS
LIN {X 69.183,Y -41.649,Z -102.611,A -90.000,B 90.000,C 0.000} C_DIS
LIN {X 69.030,Y -41.594,Z -102.377,A -90.000,B 90.000,C 0.000} C_DIS
LIN {X 68.871,Y -41.523,Z -102.127,A -90.000,B 90.000,C 0.000} C_DIS
LIN {X 68.405,Y -41.370,Z -101.413,A -90.000,B 90.000,C 0.000} C_DIS
LIN {X 68.299,Y -41.336,Z -101.246,A -90.000,B 90.000,C 0.000} C_DIS
LIN {X 68.212,Y -41.318,Z -101.110,A -90.000,B 90.000,C 0.000} C_DIS
LIN {X 68.141,Y -41.308,Z -100.999,A -90.000,B 90.000,C 0.000} C_DIS
LIN {X 68.141,Y -60.000,Z -100.999,A -90.000,B 90.000,C 0.000} C_DIS
LIN {X 84.974,Y -60.000,Z -106.902,A -90.000,B 90.000,C 0.000} C_DIS
LIN {X 84.974,Y -41.308,Z -106.902,A -90.000,B 90.000,C 0.000} C_DIS
LIN {X 84.713,Y -41.402,Z -107.048,A -90.000,B 90.000,C 0.000} C_DIS
LIN {X 84.536,Y -41.466,Z -107.144,A -90.000,B 90.000,C 0.000} C_DIS
LIN {X 84.187,Y -41.592,Z -107.315,A -90.000,B 90.000,C 0.000} C_DIS
LIN {X 83.811,Y -41.729,Z -107.480,A -90.000,B 90.000,C 0.000} C_DIS
LIN {X 83.485,Y -41.848,Z -107.608,A -90.000,B 90.000,C 0.000} C_DIS
LIN {X 83.363,Y -41.893,Z -107.651,A -90.000,B 90.000,C 0.000} C_DIS
LIN {X 83.225,Y -41.933,Z -107.698,A -90.000,B 90.000,C 0.000} C_DIS
LIN {X 82.929,Y -42.018,Z -107.790,A -90.000,B 90.000,C 0.000} C_DIS
LIN {X 82.856,Y -42.039,Z -107.820,A -90.000,B 90.000,C 0.000} C_DIS
LIN {X 82.508,Y -42.111,Z -107.960,A -90.000,B 90.000,C 0.000} C_DIS
LIN {X 82.107,Y -42.185,Z -108.117,A -90.000,B 90.000,C 0.000} C_DIS
LIN {X 81.675,Y -42.252,Z -108.284,A -90.000,B 90.000,C 0.000} C_DIS
LIN {X 81.551,Y -42.271,Z -108.329,A -90.000,B 90.000,C 0.000} C_DIS
LIN {X 81.306,Y -42.309,Z -108.423,A -90.000,B 90.000,C 0.000} C_DIS
LIN {X 81.078,Y -42.344,Z -108.502,A -90.000,B 90.000,C 0.000} C_DIS
LIN {X 80.819,Y -42.385,Z -108.587,A -90.000,B 90.000,C 0.000} C_DIS
LIN {X 80.590,Y -42.422,Z -108.657,A -90.000,B 90.000,C 0.000} C_DIS
LIN {X 80.297,Y -42.470,Z -108.736,A -90.000,B 90.000,C 0.000} C_DIS
LIN {X 79.893,Y -42.539,Z -108.827,A -90.000,B 90.000,C 0.000} C_DIS
LIN {X 79.679,Y -42.568,Z -108.871,A -90.000,B 90.000,C 0.000} C_DIS
LIN {X 79.345,Y -42.615,Z -108.928,A -90.000,B 90.000,C 0.000} C_DIS
LIN {X 79.235,Y -42.622,Z -108.945,A -90.000,B 90.000,C 0.000} C_DIS
LIN {X 78.993,Y -42.639,Z -108.977,A -90.000,B 90.000,C 0.000} C_DIS
LIN {X 78.639,Y -42.663,Z -109.014,A -90.000,B 90.000,C 0.000} C_DIS
LIN {X 78.409,Y -42.680,Z -109.031,A -90.000,B 90.000,C 0.000} C_DIS
LIN {X 78.074,Y -42.704,Z -109.045,A -90.000,B 90.000,C 0.000} C_DIS
LIN {X 77.706,Y -42.732,Z -109.050,A -90.000,B 90.000,C 0.000} C_DIS
LIN {X 77.608,Y -42.740,Z -109.049,A -90.000,B 90.000,C 0.000} C_DIS
LIN {X 77.358,Y -42.760,Z -109.041,A -90.000,B 90.000,C 0.000} C_DIS
LIN {X 77.199,Y -42.773,Z -109.034,A -90.000,B 90.000,C 0.000} C_DIS
LIN {X 76.866,Y -42.800,Z -109.010,A -90.000,B 90.000,C 0.000} C_DIS
LIN {X 76.525,Y -42.832,Z -108.976,A -90.000,B 90.000,C 0.000} C_DIS
LIN {X 76.401,Y -42.842,Z -108.962,A -90.000,B 90.000,C 0.000} C_DIS
LIN {X 76.146,Y -42.856,Z -108.928,A -90.000,B 90.000,C 0.000} C_DIS
LIN {X 75.938,Y -42.868,Z -108.895,A -90.000,B 90.000,C 0.000} C_DIS
LIN {X 75.782,Y -42.867,Z -108.866,A -90.000,B 90.000,C 0.000} C_DIS
LIN {X 75.565,Y -42.864,Z -108.824,A -90.000,B 90.000,C 0.000} C_DIS
LIN {X 75.243,Y -42.858,Z -108.752,A -90.000,B 90.000,C 0.000} C_DIS
LIN {X 75.048,Y -42.855,Z -108.702,A -90.000,B 90.000,C 0.000} C_DIS
LIN {X 74.712,Y -42.851,Z -108.605,A -90.000,B 90.000,C 0.000} C_DIS
LIN {X 74.422,Y -42.847,Z -108.513,A -90.000,B 90.000,C 0.000} C_DIS
LIN {X 74.018,Y -42.842,Z -108.378,A -90.000,B 90.000,C 0.000} C_DIS
LIN {X 73.393,Y -42.835,Z -108.188,A -90.000,B 90.000,C 0.000} C_DIS
LIN {X 73.269,Y -42.827,Z -108.150,A -90.000,B 90.000,C 0.000} C_DIS
LIN {X 73.116,Y -42.815,Z -108.102,A -90.000,B 90.000,C 0.000} C_DIS
LIN {X 72.854,Y -42.791,Z -108.013,A -90.000,B 90.000,C 0.000} C_DIS
LIN {X 72.467,Y -42.728,Z -107.871,A -90.000,B 90.000,C 0.000} C_DIS
LIN {X 72.160,Y -42.678,Z -107.744,A -90.000,B 90.000,C 0.000} C_DIS
LIN {X 71.708,Y -42.603,Z -107.540,A -90.000,B 90.000,C 0.000} C_DIS
LIN {X 71.482,Y -42.566,Z -107.429,A -90.000,B 90.000,C 0.000} C_DIS
LIN {X 71.278,Y -42.532,Z -107.323,A -90.000,B 90.000,C 0.000} C_DIS
LIN {X 71.054,Y -42.496,Z -107.197,A -90.000,B 90.000,C 0.000} C_DIS
LIN {X 70.866,Y -42.457,Z -107.087,A -90.000,B 90.000,C 0.000} C_DIS
LIN {X 70.639,Y -42.409,Z -106.944,A -90.000,B 90.000,C 0.000} C_DIS
LIN {X 70.594,Y -42.396,Z -106.914,A -90.000,B 90.000,C 0.000} C_DIS
LIN {X 70.395,Y -42.329,Z -106.778,A -90.000,B 90.000,C 0.000} C_DIS
LIN {X 70.235,Y -42.274,Z -106.661,A -90.000,B 90.000,C 0.000} C_DIS
LIN {X 69.953,Y -42.176,Z -106.446,A -90.000,B 90.000,C 0.000} C_DIS
LIN {X 69.686,Y -42.082,Z -106.224,A -90.000,B 90.000,C 0.000} C_DIS
LIN {X 69.569,Y -42.040,Z -106.123,A -90.000,B 90.000,C 0.000} C_DIS
LIN {X 69.399,Y -41.986,Z -105.973,A -90.000,B 90.000,C 0.000} C_DIS
LIN {X 69.308,Y -41.956,Z -105.888,A -90.000,B 90.000,C 0.000} C_DIS
LIN {X 69.095,Y -41.879,Z -105.684,A -90.000,B 90.000,C 0.000} C_DIS
LIN {X 68.939,Y -41.821,Z -105.527,A -90.000,B 90.000,C 0.000} C_DIS
LIN {X 68.759,Y -41.730,Z -105.332,A -90.000,B 90.000,C 0.000} C_DIS
LIN {X 68.701,Y -41.701,Z -105.267,A -90.000,B 90.000,C 0.000} C_DIS
LIN {X 68.558,Y -41.627,Z -105.097,A -90.000,B 90.000,C 0.000} C_DIS
LIN {X 68.398,Y -41.543,Z -104.897,A -90.000,B 90.000,C 0.000} C_DIS
LIN {X 68.377,Y -41.532,Z -104.868,A -90.000,B 90.000,C 0.000} C_DIS
LIN {X 68.201,Y -41.453,Z -104.638,A -90.000,B 90.000,C 0.000} C_DIS
LIN {X 67.979,Y -41.350,Z -104.325,A -90.000,B 90.000,C 0.000} C_DIS
LIN {X 67.912,Y -41.319,Z -104.223,A -90.000,B 90.000,C 0.000} C_DIS
LIN {X 67.893,Y -41.308,Z -104.192,A -90.000,B 90.000,C 0.000} C_DIS
LIN {X 67.893,Y -60.000,Z -104.192,A -90.000,B 90.000,C 0.000} C_DIS
LIN {X 84.697,Y -60.000,Z -109.238,A -90.000,B 90.000,C 0.000} C_DIS
LIN {X 84.697,Y -41.308,Z -109.238,A -90.000,B 90.000,C 0.000} C_DIS
LIN {X 84.421,Y -41.387,Z -109.354,A -90.000,B 90.000,C 0.000} C_DIS
LIN {X 84.022,Y -41.503,Z -109.503,A -90.000,B 90.000,C 0.000} C_DIS
LIN {X 83.720,Y -41.592,Z -109.605,A -90.000,B 90.000,C 0.000} C_DIS
LIN {X 83.506,Y -41.656,Z -109.672,A -90.000,B 90.000,C 0.000} C_DIS
LIN {X 82.935,Y -41.820,Z -109.910,A -90.000,B 90.000,C 0.000} C_DIS
LIN {X 82.411,Y -41.946,Z -110.120,A -90.000,B 90.000,C 0.000} C_DIS
LIN {X 82.052,Y -42.000,Z -110.255,A -90.000,B 90.000,C 0.000} C_DIS
LIN {X 81.912,Y -42.020,Z -110.307,A -90.000,B 90.000,C 0.000} C_DIS
LIN {X 81.615,Y -42.064,Z -110.408,A -90.000,B 90.000,C 0.000} C_DIS
LIN {X 81.352,Y -42.100,Z -110.494,A -90.000,B 90.000,C 0.000} C_DIS
LIN {X 81.062,Y -42.140,Z -110.580,A -90.000,B 90.000,C 0.000} C_DIS
LIN {X 80.768,Y -42.181,Z -110.658,A -90.000,B 90.000,C 0.000} C_DIS
LIN {X 80.669,Y -42.196,Z -110.682,A -90.000,B 90.000,C 0.000} C_DIS
LIN {X 80.250,Y -42.257,Z -110.775,A -90.000,B 90.000,C 0.000} C_DIS
LIN {X 79.978,Y -42.298,Z -110.830,A -90.000,B 90.000,C 0.000} C_DIS
LIN {X 79.483,Y -42.374,Z -110.914,A -90.000,B 90.000,C 0.000} C_DIS
LIN {X 79.188,Y -42.421,Z -110.955,A -90.000,B 90.000,C 0.000} C_DIS
LIN {X 78.872,Y -42.464,Z -110.991,A -90.000,B 90.000,C 0.000} C_DIS
LIN {X 78.655,Y -42.495,Z -111.010,A -90.000,B 90.000,C 0.000} C_DIS
LIN {X 78.554,Y -42.502,Z -111.017,A -90.000,B 90.000,C 0.000} C_DIS
LIN {X 78.089,Y -42.533,Z -111.038,A -90.000,B 90.000,C 0.000} C_DIS
LIN {X 77.668,Y -42.562,Z -111.043,A -90.000,B 90.000,C 0.000} C_DIS
LIN {X 77.471,Y -42.576,Z -111.039,A -90.000,B 90.000,C 0.000} C_DIS
LIN {X 77.045,Y -42.608,Z -111.021,A -90.000,B 90.000,C 0.000} C_DIS
LIN {X 76.637,Y -42.640,Z -110.991,A -90.000,B 90.000,C 0.000} C_DIS
LIN {X 76.281,Y -42.669,Z -110.954,A -90.000,B 90.000,C 0.000} C_DIS
LIN {X 76.203,Y -42.675,Z -110.945,A -90.000,B 90.000,C 0.000} C_DIS
LIN {X 75.821,Y -42.708,Z -110.896,A -90.000,B 90.000,C 0.000} C_DIS
LIN {X 75.507,Y -42.735,Z -110.845,A -90.000,B 90.000,C 0.000} C_DIS
LIN {X 75.129,Y -42.755,Z -110.773,A -90.000,B 90.000,C 0.000} C_DIS
LIN {X 75.039,Y -42.759,Z -110.753,A -90.000,B 90.000,C 0.000} C_DIS
LIN {X 74.852,Y -42.758,Z -110.711,A -90.000,B 90.000,C 0.000} C_DIS
LIN {X 74.728,Y -42.756,Z -110.682,A -90.000,B 90.000,C 0.000} C_DIS
LIN {X 74.498,Y -42.754,Z -110.622,A -90.000,B 90.000,C 0.000} C_DIS
LIN {X 74.108,Y -42.750,Z -110.509,A -90.000,B 90.000,C 0.000} C_DIS
LIN {X 73.762,Y -42.746,Z -110.399,A -90.000,B 90.000,C 0.000} C_DIS
LIN {X 73.384,Y -42.743,Z -110.273,A -90.000,B 90.000,C 0.000} C_DIS
LIN {X 72.556,Y -42.733,Z -110.021,A -90.000,B 90.000,C 0.000} C_DIS
LIN {X 72.325,Y -42.730,Z -109.944,A -90.000,B 90.000,C 0.000} C_DIS
LIN {X 72.212,Y -42.722,Z -109.906,A -90.000,B 90.000,C 0.000} C_DIS
LIN {X 71.833,Y -42.691,Z -109.768,A -90.000,B 90.000,C 0.000} C_DIS
LIN {X 71.729,Y -42.673,Z -109.729,A -90.000,B 90.000,C 0.000} C_DIS
LIN {X 71.332,Y -42.606,Z -109.564,A -90.000,B 90.000,C 0.000} C_DIS
LIN {X 70.835,Y -42.522,Z -109.338,A -90.000,B 90.000,C 0.000} C_DIS
LIN {X 70.641,Y -42.489,Z -109.242,A -90.000,B 90.000,C 0.000} C_DIS
LIN {X 70.372,Y -42.444,Z -109.104,A -90.000,B 90.000,C 0.000} C_DIS
LIN {X 70.023,Y -42.385,Z -108.908,A -90.000,B 90.000,C 0.000} C_DIS
LIN {X 69.895,Y -42.361,Z -108.833,A -90.000,B 90.000,C 0.000} C_DIS
LIN {X 69.654,Y -42.310,Z -108.683,A -90.000,B 90.000,C 0.000} C_DIS
LIN {X 69.514,Y -42.278,Z -108.594,A -90.000,B 90.000,C 0.000} C_DIS
LIN {X 69.362,Y -42.224,Z -108.489,A -90.000,B 90.000,C 0.000} C_DIS
LIN {X 69.142,Y -42.145,Z -108.332,A -90.000,B 90.000,C 0.000} C_DIS
LIN {X 68.752,Y -42.000,Z -108.035,A -90.000,B 90.000,C 0.000} C_DIS
LIN {X 68.645,Y -41.959,Z -107.947,A -90.000,B 90.000,C 0.000} C_DIS
LIN {X 68.423,Y -41.880,Z -107.761,A -90.000,B 90.000,C 0.000} C_DIS
LIN {X 68.103,Y -41.766,Z -107.480,A -90.000,B 90.000,C 0.000} C_DIS
LIN {X 67.855,Y -41.673,Z -107.244,A -90.000,B 90.000,C 0.000} C_DIS
LIN {X 67.710,Y -41.595,Z -107.099,A -90.000,B 90.000,C 0.000} C_DIS
LIN {X 67.603,Y -41.536,Z -106.988,A -90.000,B 90.000,C 0.000} C_DIS
LIN {X 67.469,Y -41.462,Z -106.843,A -90.000,B 90.000,C 0.000} C_DIS
LIN {X 67.322,Y -41.387,Z -106.680,A -90.000,B 90.000,C 0.000} C_DIS
LIN {X 67.169,Y -41.308,Z -106.502,A -90.000,B 90.000,C 0.000} C_DIS
LIN {X 67.169,Y -60.000,Z -106.502,A -90.000,B 90.000,C 0.000} C_DIS
LIN {X 54.853,Y -60.000,Z -129.945,A -90.000,B 90.000,C 0.000} C_DIS
LIN {X 54.853,Y -41.308,Z -129.945,A -90.000,B 90.000,C 0.000} C_DIS
LIN {X 55.546,Y -41.380,Z -129.212,A -90.000,B 90.000,C 0.000} C_DIS
LIN {X 56.167,Y -41.439,Z -128.533,A -90.000,B 90.000,C 0.000} C_DIS
LIN {X 57.160,Y -41.453,Z -127.023,A -90.000,B 90.000,C 0.000} C_DIS
LIN {X 57.408,Y -41.463,Z -126.642,A -90.000,B 90.000,C 0.000} C_DIS
LIN {X 58.229,Y -41.499,Z -125.406,A -90.000,B 90.000,C 0.000} C_DIS
LIN {X 58.695,Y -41.509,Z -124.640,A -90.000,B 90.000,C 0.000} C_DIS
LIN {X 58.911,Y -41.518,Z -124.287,A -90.000,B 90.000,C 0.000} C_DIS
LIN {X 59.030,Y -41.526,Z -124.106,A -90.000,B 90.000,C 0.000} C_DIS
LIN {X 59.133,Y -41.533,Z -123.960,A -90.000,B 90.000,C 0.000} C_DIS
LIN {X 59.252,Y -41.544,Z -123.803,A -90.000,B 90.000,C 0.000} C_DIS
LIN {X 59.375,Y -41.557,Z -123.648,A -90.000,B 90.000,C 0.000} C_DIS
LIN {X 59.554,Y -41.577,Z -123.435,A -90.000,B 90.000,C 0.000} C_DIS
LIN {X 59.692,Y -41.587,Z -123.278,A -90.000,B 90.000,C 0.000} C_DIS
LIN {X 59.856,Y -41.602,Z -123.105,A -90.000,B 90.000,C 0.000} C_DIS
LIN {X 60.016,Y -41.617,Z -122.947,A -90.000,B 90.000,C 0.000} C_DIS
LIN {X 60.256,Y -41.641,Z -122.715,A -90.000,B 90.000,C 0.000} C_DIS
LIN {X 60.603,Y -41.660,Z -122.291,A -90.000,B 90.000,C 0.000} C_DIS
LIN {X 61.315,Y -41.731,Z -121.405,A -90.000,B 90.000,C 0.000} C_DIS
LIN {X 61.646,Y -41.766,Z -121.011,A -90.000,B 90.000,C 0.000} C_DIS
LIN {X 61.795,Y -41.784,Z -120.847,A -90.000,B 90.000,C 0.000} C_DIS
LIN {X 61.941,Y -41.803,Z -120.698,A -90.000,B 90.000,C 0.000} C_DIS
LIN {X 62.120,Y -41.828,Z -120.529,A -90.000,B 90.000,C 0.000} C_DIS
LIN {X 62.255,Y -41.847,Z -120.406,A -90.000,B 90.000,C 0.000} C_DIS
LIN {X 62.583,Y -41.897,Z -120.138,A -90.000,B 90.000,C 0.000} C_DIS
LIN {X 62.720,Y -41.919,Z -120.031,A -90.000,B 90.000,C 0.000} C_DIS
LIN {X 62.880,Y -41.941,Z -119.916,A -90.000,B 90.000,C 0.000} C_DIS
LIN {X 62.970,Y -41.948,Z -119.855,A -90.000,B 90.000,C 0.000} C_DIS
LIN {X 63.081,Y -41.957,Z -119.783,A -90.000,B 90.000,C 0.000} C_DIS
LIN {X 63.136,Y -41.960,Z -119.749,A -90.000,B 90.000,C 0.000} C_DIS
LIN {X 63.290,Y -41.979,Z -119.655,A -90.000,B 90.000,C 0.000} C_DIS
LIN {X 63.479,Y -42.003,Z -119.549,A -90.000,B 90.000,C 0.000} C_DIS
LIN {X 65.109,Y -42.214,Z -118.703,A -90.000,B 90.000,C 0.000} C_DIS
LIN {X 65.479,Y -42.261,Z -118.512,A -90.000,B 90.000,C 0.000} C_DIS
LIN {X 65.647,Y -42.280,Z -118.386,A -90.000,B 90.000,C 0.000} C_DIS
LIN {X 65.795,Y -42.297,Z -118.283,A -90.000,B 90.000,C 0.000} C_DIS
LIN {X 65.940,Y -42.314,Z -118.187,A -90.000,B 90.000,C 0.000} C_DIS
LIN {X 66.134,Y -42.337,Z -118.068,A -90.000,B 90.000,C 0.000} C_DIS
LIN {X 66.369,Y -42.366,Z -117.931,A -90.000,B 90.000,C 0.000} C_DIS
LIN {X 66.591,Y -42.394,Z -117.812,A -90.000,B 90.000,C 0.000} C_DIS
LIN {X 66.737,Y -42.413,Z -117.739,A -90.000,B 90.000,C 0.000} C_DIS
LIN {X 66.827,Y -42.425,Z -117.697,A -90.000,B 90.000,C 0.000} C_DIS
LIN {X 66.994,Y -42.447,Z -117.625,A -90.000,B 90.000,C 0.000} C_DIS
LIN {X 67.208,Y -42.476,Z -117.539,A -90.000,B 90.000,C 0.000} C_DIS
LIN {X 67.329,Y -42.488,Z -117.498,A -90.000,B 90.000,C 0.000} C_DIS
LIN {X 67.447,Y -42.495,Z -117.459,A -90.000,B 90.000,C 0.000} C_DIS
LIN {X 67.648,Y -42.499,Z -117.400,A -90.000,B 90.000,C 0.000} C_DIS
LIN {X 67.828,Y -42.497,Z -117.355,A -90.000,B 90.000,C 0.000} C_DIS
LIN {X 68.024,Y -42.492,Z -117.309,A -90.000,B 90.000,C 0.000} C_DIS
LIN {X 68.297,Y -42.486,Z -117.253,A -90.000,B 90.000,C 0.000} C_DIS
LIN {X 68.449,Y -42.486,Z -117.227,A -90.000,B 90.000,C 0.000} C_DIS
LIN {X 68.643,Y -42.489,Z -117.200,A -90.000,B 90.000,C 0.000} C_DIS
LIN {X 68.712,Y -42.490,Z -117.193,A -90.000,B 90.000,C 0.000} C_DIS
LIN {X 68.857,Y -42.492,Z -117.182,A -90.000,B 90.000,C 0.000} C_DIS
LIN {X 69.295,Y -42.500,Z -117.160,A -90.000,B 90.000,C 0.000} C_DIS
LIN {X 69.545,Y -42.506,Z -117.158,A -90.000,B 90.000,C 0.000} C_DIS
LIN {X 69.854,Y -42.513,Z -117.169,A -90.000,B 90.000,C 0.000} C_DIS
LIN {X 70.138,Y -42.520,Z -117.190,A -90.000,B 90.000,C 0.000} C_DIS
LIN {X 70.346,Y -42.526,Z -117.209,A -90.000,B 90.000,C 0.000} C_DIS
LIN {X 70.738,Y -42.537,Z -117.264,A -90.000,B 90.000,C 0.000} C_DIS
LIN {X 71.045,Y -42.547,Z -117.322,A -90.000,B 90.000,C 0.000} C_DIS
LIN {X 72.017,Y -42.579,Z -117.526,A -90.000,B 90.000,C 0.000} C_DIS
LIN {X 72.332,Y -42.590,Z -117.599,A -90.000,B 90.000,C 0.000} C_DIS
LIN {X 72.457,Y -42.587,Z -117.629,A -90.000,B 90.000,C 0.000} C_DIS
LIN {X 72.862,Y -42.566,Z -117.727,A -90.000,B 90.000,C 0.000} C_DIS
LIN {X 73.031,Y -42.552,Z -117.770,A -90.000,B 90.000,C 0.000} C_DIS
LIN {X 73.334,Y -42.528,Z -117.860,A -90.000,B 90.000,C 0.000} C_DIS
LIN {X 73.700,Y -42.499,Z -117.987,A -90.000,B 90.000,C 0.000} C_DIS
LIN {X 73.809,Y -42.491,Z -118.026,A -90.000,B 90.000,C 0.000} C_DIS
LIN {X 75.907,Y -42.332,Z -118.839,A -90.000,B 90.000,C 0.000} C_DIS
LIN {X 76.030,Y -42.324,Z -118.894,A -90.000,B 90.000,C 0.000} C_DIS
LIN {X 76.223,Y -42.310,Z -118.989,A -90.000,B 90.000,C 0.000} C_DIS
LIN {X 76.713,Y -42.284,Z -119.252,A -90.000,B 90.000,C 0.000} C_DIS
LIN {X 76.870,Y -42.277,Z -119.346,A -90.000,B 90.000,C 0.000} C_DIS
LIN {X 76.951,Y -42.273,Z -119.397,A -90.000,B 90.000,C 0.000} C_DIS
LIN {X 77.144,Y -42.253,Z -119.532,A -90.000,B 90.000,C 0.000} C_DIS
LIN {X 77.479,Y -42.218,Z -119.777,A -90.000,B 90.000,C 0.000} C_DIS
LIN {X 77.830,Y -42.170,Z -120.043,A -90.000,B 90.000,C 0.000} C_DIS
LIN {X 77.901,Y -42.161,Z -120.099,A -90.000,B 90.000,C 0.000} C_DIS
LIN {X 78.130,Y -42.131,Z -120.292,A -90.000,B 90.000,C 0.000} C_DIS
LIN {X 78.300,Y -42.111,Z -120.448,A -90.000,B 90.000,C 0.000} C_DIS
LIN {X 78.455,Y -42.093,Z -120.603,A -90.000,B 90.000,C 0.000} C_DIS
LIN {X 78.656,Y -42.071,Z -120.812,A -90.000,B 90.000,C 0.000} C_DIS
LIN {X 78.885,Y -42.047,Z -121.069,A -90.000,B 90.000,C 0.000} C_DIS
LIN {X 78.961,Y -42.038,Z -121.156,A -90.000,B 90.000,C 0.000} C_DIS
LIN {X 79.106,Y -42.023,Z -121.334,A -90.000,B 90.000,C 0.000} C_DIS
LIN {X 79.312,Y -42.002,Z -121.605,A -90.000,B 90.000,C 0.000} C_DIS
LIN {X 79.356,Y -41.998,Z -121.667,A -90.000,B 90.000,C 0.000} C_DIS
LIN {X 79.616,Y -41.976,Z -122.053,A -90.000,B 90.000,C 0.000} C_DIS
LIN {X 80.282,Y -41.949,Z -123.046,A -90.000,B 90.000,C 0.000} C_DIS
LIN {X 80.403,Y -41.936,Z -123.231,A -90.000,B 90.000,C 0.000} C_DIS
LIN {X 80.578,Y -41.919,Z -123.526,A -90.000,B 90.000,C 0.000} C_DIS
LIN {X 80.740,Y -41.905,Z -123.812,A -90.000,B 90.000,C 0.000} C_DIS
LIN {X 80.864,Y -41.895,Z -124.055,A -90.000,B 90.000,C 0.000} C_DIS
LIN {X 80.925,Y -41.892,Z -124.184,A -90.000,B 90.000,C 0.000} C_DIS
LIN {X 81.039,Y -41.887,Z -124.455,A -90.000,B 90.000,C 0.000} C_DIS
LIN {X 81.075,Y -41.886,Z -124.542,A -90.000,B 90.000,C 0.000} C_DIS
LIN {X 81.122,Y -41.885,Z -124.669,A -90.000,B 90.000,C 0.000} C_DIS
LIN {X 81.249,Y -41.893,Z -124.999,A -90.000,B 90.000,C 0.000} C_DIS
LIN {X 81.320,Y -41.891,Z -125.194,A -90.000,B 90.000,C 0.000} C_DIS
LIN {X 81.396,Y -41.889,Z -125.408,A -90.000,B 90.000,C 0.000} C_DIS
LIN {X 81.719,Y -41.839,Z -126.351,A -90.000,B 90.000,C 0.000} C_DIS
LIN {X 81.814,Y -41.825,Z -126.651,A -90.000,B 90.000,C 0.000} C_DIS
LIN {X 81.904,Y -41.813,Z -126.979,A -90.000,B 90.000,C 0.000} C_DIS
LIN {X 81.946,Y -41.807,Z -127.149,A -90.000,B 90.000,C 0.000} C_DIS
LIN {X 81.972,Y -41.803,Z -127.270,A -90.000,B 90.000,C 0.000} C_DIS
LIN {X 82.121,Y -41.769,Z -128.118,A -90.000,B 90.000,C 0.000} C_DIS
LIN {X 82.158,Y -41.761,Z -128.345,A -90.000,B 90.000,C 0.000} C_DIS
LIN {X 82.257,Y -41.740,Z -129.038,A -90.000,B 90.000,C 0.000} C_DIS
LIN {X 82.294,Y -41.727,Z -129.310,A -90.000,B 90.000,C 0.000} C_DIS
LIN {X 82.319,Y -41.716,Z -129.509,A -90.000,B 90.000,C 0.000} C_DIS
LIN {X 82.364,Y -41.695,Z -129.972,A -90.000,B 90.000,C 0.000} C_DIS
LIN {X 82.444,Y -41.654,Z -131.072,A -90.000,B 90.000,C 0.000} C_DIS
LIN {X 82.471,Y -41.640,Z -131.371,A -90.000,B 90.000,C 0.000} C_DIS
LIN {X 82.490,Y -41.626,Z -131.587,A -90.000,B 90.000,C 0.000} C_DIS
LIN {X 82.533,Y -41.603,Z -132.088,A -90.000,B 90.000,C 0.000} C_DIS
LIN {X 82.612,Y -41.555,Z -133.506,A -90.000,B 90.000,C 0.000} C_DIS
LIN {X 82.675,Y -41.511,Z -134.225,A -90.000,B 90.000,C 0.000} C_DIS
LIN {X 82.713,Y -41.490,Z -134.652,A -90.000,B 90.000,C 0.000} C_DIS
LIN {X 82.774,Y -41.462,Z -135.312,A -90.000,B 90.000,C 0.000} C_DIS
LIN {X 82.841,Y -41.430,Z -135.837,A -90.000,B 90.000,C 0.000} C_DIS
LIN {X 82.942,Y -41.383,Z -136.878,A -90.000,B 90.000,C 0.000} C_DIS
LIN {X 82.978,Y -41.363,Z -137.276,A -90.000,B 90.000,C 0.000} C_DIS
LIN {X 83.071,Y -41.308,Z -138.307,A -90.000,B 90.000,C 0.000} C_DIS
LIN {X 83.071,Y -60.000,Z -138.307,A -90.000,B 90.000,C 0.000} C_DIS
LIN {X 61.279,Y -60.000,Z -118.728,A -90.000,B 90.000,C 0.000} C_DIS
LIN {X 61.279,Y -41.308,Z -118.728,A -90.000,B 90.000,C 0.000} C_DIS
LIN {X 61.491,Y -41.345,Z -118.555,A -90.000,B 90.000,C 0.000} C_DIS
LIN {X 61.651,Y -41.374,Z -118.431,A -90.000,B 90.000,C 0.000} C_DIS
LIN {X 61.939,Y -41.429,Z -118.222,A -90.000,B 90.000,C 0.000} C_DIS
LIN {X 62.123,Y -41.465,Z -118.097,A -90.000,B 90.000,C 0.000} C_DIS
LIN {X 62.330,Y -41.507,Z -117.965,A -90.000,B 90.000,C 0.000} C_DIS
LIN {X 62.624,Y -41.569,Z -117.794,A -90.000,B 90.000,C 0.000} C_DIS
LIN {X 63.149,Y -41.684,Z -117.510,A -90.000,B 90.000,C 0.000} C_DIS
LIN {X 63.793,Y -41.805,Z -117.168,A -90.000,B 90.000,C 0.000} C_DIS
LIN {X 64.461,Y -41.898,Z -116.821,A -90.000,B 90.000,C 0.000} C_DIS
LIN {X 64.605,Y -41.914,Z -116.717,A -90.000,B 90.000,C 0.000} C_DIS
LIN {X 64.776,Y -41.935,Z -116.599,A -90.000,B 90.000,C 0.000} C_DIS
LIN {X 64.946,Y -41.956,Z -116.488,A -90.000,B 90.000,C 0.000} C_DIS
LIN {X 65.205,Y -41.989,Z -116.331,A -90.000,B 90.000,C 0.000} C_DIS
LIN {X 65.471,Y -42.024,Z -116.176,A -90.000,B 90.000,C 0.000} C_DIS
LIN {X 65.748,Y -42.062,Z -116.028,A -90.000,B 90.000,C 0.000} C_DIS
LIN {X 65.980,Y -42.095,Z -115.915,A -90.000,B 90.000,C 0.000} C_DIS
LIN {X 66.184,Y -42.125,Z -115.824,A -90.000,B 90.000,C 0.000} C_DIS
LIN {X 66.297,Y -42.142,Z -115.775,A -90.000,B 90.000,C 0.000} C_DIS
LIN {X 66.587,Y -42.187,Z -115.660,A -90.000,B 90.000,C 0.000} C_DIS
LIN {X 66.894,Y -42.236,Z -115.554,A -90.000,B 90.000,C 0.000} C_DIS
LIN {X 67.160,Y -42.279,Z -115.473,A -90.000,B 90.000,C 0.000} C_DIS
LIN {X 67.374,Y -42.315,Z -115.416,A -90.000,B 90.000,C 0.000} C_DIS
LIN {X 67.646,Y -42.361,Z -115.349,A -90.000,B 90.000,C 0.000} C_DIS
LIN {X 67.666,Y -42.364,Z -115.345,A -90.000,B 90.000,C 0.000} C_DIS
LIN {X 67.960,Y -42.407,Z -115.283,A -90.000,B 90.000,C 0.000} C_DIS
LIN {X 68.172,Y -42.439,Z -115.247,A -90.000,B 90.000,C 0.000} C_DIS
LIN {X 68.302,Y -42.459,Z -115.229,A -90.000,B 90.000,C 0.000} C_DIS
LIN {X 68.502,Y -42.474,Z -115.204,A -90.000,B 90.000,C 0.000} C_DIS
LIN {X 68.797,Y -42.496,Z -115.182,A -90.000,B 90.000,C 0.000} C_DIS
LIN {X 68.924,Y -42.505,Z -115.176,A -90.000,B 90.000,C 0.000} C_DIS
LIN {X 69.158,Y -42.510,Z -115.165,A -90.000,B 90.000,C 0.000} C_DIS
LIN {X 69.288,Y -42.512,Z -115.160,A -90.000,B 90.000,C 0.000} C_DIS
LIN {X 69.525,Y -42.515,Z -115.158,A -90.000,B 90.000,C 0.000} C_DIS
LIN {X 69.653,Y -42.517,Z -115.160,A -90.000,B 90.000,C 0.000} C_DIS
LIN {X 70.000,Y -42.522,Z -115.175,A -90.000,B 90.000,C 0.000} C_DIS
LIN {X 70.484,Y -42.529,Z -115.213,A -90.000,B 90.000,C 0.000} C_DIS
LIN {X 70.617,Y -42.531,Z -115.227,A -90.000,B 90.000,C 0.000} C_DIS
LIN {X 71.017,Y -42.536,Z -115.283,A -90.000,B 90.000,C 0.000} C_DIS
LIN {X 71.212,Y -42.539,Z -115.318,A -90.000,B 90.000,C 0.000} C_DIS
LIN {X 71.442,Y -42.542,Z -115.362,A -90.000,B 90.000,C 0.000} C_DIS
LIN {X 72.473,Y -42.557,Z -115.578,A -90.000,B 90.000,C 0.000} C_DIS
LIN {X 72.832,Y -42.561,Z -115.663,A -90.000,B 90.000,C 0.000} C_DIS
LIN {X 72.922,Y -42.559,Z -115.684,A -90.000,B 90.000,C 0.000} C_DIS
LIN {X 73.510,Y -42.510,Z -115.829,A -90.000,B 90.000,C 0.000} C_DIS
LIN {X 73.594,Y -42.503,Z -115.852,A -90.000,B 90.000,C 0.000} C_DIS
LIN {X 73.966,Y -42.472,Z -115.963,A -90.000,B 90.000,C 0.000} C_DIS
LIN {X 74.377,Y -42.435,Z -116.106,A -90.000,B 90.000,C 0.000} C_DIS
LIN {X 74.539,Y -42.421,Z -116.166,A -90.000,B 90.000,C 0.000} C_DIS
LIN {X 76.621,Y -42.220,Z -116.974,A -90.000,B 90.000,C 0.000} C_DIS
LIN {X 76.777,Y -42.206,Z -117.042,A -90.000,B 90.000,C 0.000} C_DIS
LIN {X 76.901,Y -42.197,Z -117.098,A -90.000,B 90.000,C 0.000} C_DIS
LIN {X 77.046,Y -42.187,Z -117.170,A -90.000,B 90.000,C 0.000} C_DIS
LIN {X 77.187,Y -42.163,Z -117.243,A -90.000,B 90.000,C 0.000} C_DIS
LIN {X 77.647,Y -42.085,Z -117.495,A -90.000,B 90.000,C 0.000} C_DIS
LIN {X 77.756,Y -42.066,Z -117.559,A -90.000,B 90.000,C 0.000} C_DIS
LIN {X 77.879,Y -42.045,Z -117.634,A -90.000,B 90.000,C 0.000} C_DIS
LIN {X 78.067,Y -42.014,Z -117.758,A -90.000,B 90.000,C 0.000} C_DIS
LIN {X 78.258,Y -41.982,Z -117.893,A -90.000,B 90.000,C 0.000} C_DIS
LIN {X 78.707,Y -41.908,Z -118.227,A -90.000,B 90.000,C 0.000} C_DIS
LIN {X 79.032,Y -41.854,Z -118.476,A -90.000,B 90.000,C 0.000} C_DIS
LIN {X 79.179,Y -41.830,Z -118.596,A -90.000,B 90.000,C 0.000} C_DIS
LIN {X 79.375,Y -41.798,Z -118.762,A -90.000,B 90.000,C 0.000} C_DIS
LIN {X 79.440,Y -41.787,Z -118.820,A -90.000,B 90.000,C 0.000} C_DIS
LIN {X 79.672,Y -41.750,Z -119.038,A -90.000,B 90.000,C 0.000} C_DIS
LIN {X 79.855,Y -41.721,Z -119.224,A -90.000,B 90.000,C 0.000} C_DIS
LIN {X 80.102,Y -41.689,Z -119.485,A -90.000,B 90.000,C 0.000} C_DIS
LIN {X 80.430,Y -41.648,Z -119.856,A -90.000,B 90.000,C 0.000} C_DIS
LIN {X 80.656,Y -41.621,Z -120.136,A -90.000,B 90.000,C 0.000} C_DIS
LIN {X 80.886,Y -41.594,Z -120.441,A -90.000,B 90.000,C 0.000} C_DIS
LIN {X 80.972,Y -41.584,Z -120.563,A -90.000,B 90.000,C 0.000} C_DIS
LIN {X 81.416,Y -41.537,Z -121.232,A -90.000,B 90.000,C 0.000} C_DIS
LIN {X 81.947,Y -41.456,Z -122.048,A -90.000,B 90.000,C 0.000} C_DIS
LIN {X 82.054,Y -41.437,Z -122.219,A -90.000,B 90.000,C 0.000} C_DIS
LIN {X 82.252,Y -41.404,Z -122.559,A -90.000,B 90.000,C 0.000} C_DIS
LIN {X 82.410,Y -41.378,Z -122.847,A -90.000,B 90.000,C 0.000} C_DIS
LIN {X 82.513,Y -41.363,Z -123.049,A -90.000,B 90.000,C 0.000} C_DIS
LIN {X 82.593,Y -41.351,Z -123.210,A -90.000,B 90.000,C 0.000} C_DIS
LIN {X 82.656,Y -41.337,Z -123.349,A -90.000,B 90.000,C 0.000} C_DIS
LIN {X 82.751,Y -41.317,Z -123.582,A -90.000,B 90.000,C 0.000} C_DIS
LIN {X 82.815,Y -41.308,Z -123.740,A -90.000,B 90.000,C 0.000} C_DIS
LIN {X 82.815,Y -60.000,Z -123.740,A -90.000,B 90.000,C 0.000} C_DIS
LIN {X 63.041,Y -60.000,Z -115.380,A -90.000,B 90.000,C 0.000} C_DIS
LIN {X 63.041,Y -41.308,Z -115.380,A -90.000,B 90.000,C 0.000} C_DIS
LIN {X 63.486,Y -41.409,Z -115.138,A -90.000,B 90.000,C 0.000} C_DIS
LIN {X 63.754,Y -41.462,Z -114.947,A -90.000,B 90.000,C 0.000} C_DIS
LIN {X 63.976,Y -41.508,Z -114.797,A -90.000,B 90.000,C 0.000} C_DIS
LIN {X 64.264,Y -41.570,Z -114.616,A -90.000,B 90.000,C 0.000} C_DIS
LIN {X 64.587,Y -41.642,Z -114.424,A -90.000,B 90.000,C 0.000} C_DIS
LIN {X 64.849,Y -41.701,Z -114.279,A -90.000,B 90.000,C 0.000} C_DIS
LIN {X 65.047,Y -41.742,Z -114.177,A -90.000,B 90.000,C 0.000} C_DIS
LIN {X 65.204,Y -41.774,Z -114.100,A -90.000,B 90.000,C 0.000} C_DIS
LIN {X 65.545,Y -41.847,Z -113.946,A -90.000,B 90.000,C 0.000} C_DIS
LIN {X 65.817,Y -41.906,Z -113.834,A -90.000,B 90.000,C 0.000} C_DIS
LIN {X 65.993,Y -41.934,Z -113.767,A -90.000,B 90.000,C 0.000} C_DIS
LIN {X 66.349,Y -41.992,Z -113.646,A -90.000,B 90.000,C 0.000} C_DIS
LIN {X 66.619,Y -42.036,Z -113.563,A -90.000,B 90.000,C 0.000} C_DIS
LIN {X 66.929,Y -42.083,Z -113.479,A -90.000,B 90.000,C 0.000} C_DIS
LIN {X 67.292,Y -42.138,Z -113.393,A -90.000,B 90.000,C 0.000} C_DIS
LIN {X 67.655,Y -42.194,Z -113.318,A -90.000,B 90.000,C 0.000} C_DIS
LIN {X 67.927,Y -42.236,Z -113.272,A -90.000,B 90.000,C 0.000} C_DIS
LIN {X 68.318,Y -42.297,Z -113.220,A -90.000,B 90.000,C 0.000} C_DIS
LIN {X 68.708,Y -42.359,Z -113.189,A -90.000,B 90.000,C 0.000} C_DIS
LIN {X 69.087,Y -42.418,Z -113.168,A -90.000,B 90.000,C 0.000} C_DIS
LIN {X 69.269,Y -42.446,Z -113.161,A -90.000,B 90.000,C 0.000} C_DIS
LIN {X 69.566,Y -42.493,Z -113.158,A -90.000,B 90.000,C 0.000} C_DIS
LIN {X 69.693,Y -42.512,Z -113.161,A -90.000,B 90.000,C 0.000} C_DIS
LIN {X 70.082,Y -42.546,Z -113.177,A -90.000,B 90.000,C 0.000} C_DIS
LIN {X 70.255,Y -42.561,Z -113.189,A -90.000,B 90.000,C 0.000} C_DIS
LIN {X 70.364,Y -42.565,Z -113.198,A -90.000,B 90.000,C 0.000} C_DIS
LIN {X 70.700,Y -42.571,Z -113.225,A -90.000,B 90.000,C 0.000} C_DIS
LIN {X 70.910,Y -42.575,Z -113.249,A -90.000,B 90.000,C 0.000} C_DIS
LIN {X 71.366,Y -42.581,Z -113.315,A -90.000,B 90.000,C 0.000} C_DIS
LIN {X 71.701,Y -42.585,Z -113.376,A -90.000,B 90.000,C 0.000} C_DIS
LIN {X 71.970,Y -42.588,Z -113.430,A -90.000,B 90.000,C 0.000} C_DIS
LIN {X 72.929,Y -42.598,Z -113.632,A -90.000,B 90.000,C 0.000} C_DIS
LIN {X 73.502,Y -42.604,Z -113.768,A -90.000,B 90.000,C 0.000} C_DIS
LIN {X 73.591,Y -42.603,Z -113.790,A -90.000,B 90.000,C 0.000} C_DIS
LIN {X 74.029,Y -42.575,Z -113.899,A -90.000,B 90.000,C 0.000} C_DIS
LIN {X 74.200,Y -42.559,Z -113.947,A -90.000,B 90.000,C 0.000} C_DIS
LIN {X 74.626,Y -42.518,Z -114.076,A -90.000,B 90.000,C 0.000} C_DIS
LIN {X 75.104,Y -42.470,Z -114.243,A -90.000,B 90.000,C 0.000} C_DIS
LIN {X 75.233,Y -42.458,Z -114.290,A -90.000,B 90.000,C 0.000} C_DIS
LIN {X 76.251,Y -42.354,Z -114.685,A -90.000,B 90.000,C 0.000} C_DIS
LIN {X 77.100,Y -42.277,Z -115.015,A -90.000,B 90.000,C 0.000} C_DIS
LIN {X 77.415,Y -42.246,Z -115.139,A -90.000,B 90.000,C 0.000} C_DIS
LIN {X 77.451,Y -42.243,Z -115.154,A -90.000,B 90.000,C 0.000} C_DIS
LIN {X 77.673,Y -42.200,Z -115.252,A -90.000,B 90.000,C 0.000} C_DIS
LIN {X 77.736,Y -42.188,Z -115.281,A -90.000,B 90.000,C 0.000} C_DIS
LIN {X 77.961,Y -42.144,Z -115.391,A -90.000,B 90.000,C 0.000} C_DIS
LIN {X 78.142,Y -42.109,Z -115.486,A -90.000,B 90.000,C 0.000} C_DIS
LIN {X 78.652,Y -42.007,Z -115.768,A -90.000,B 90.000,C 0.000} C_DIS
LIN {X 78.959,Y -41.945,Z -115.954,A -90.000,B 90.000,C 0.000} C_DIS
LIN {X 79.126,Y -41.911,Z -116.064,A -90.000,B 90.000,C 0.000} C_DIS
LIN {X 79.297,Y -41.874,Z -116.183,A -90.000,B 90.000,C 0.000} C_DIS
LIN {X 79.435,Y -41.845,Z -116.282,A -90.000,B 90.000,C 0.000} C_DIS
LIN {X 79.952,Y -41.734,Z -116.670,A -90.000,B 90.000,C 0.000} C_DIS
LIN {X 80.274,Y -41.664,Z -116.920,A -90.000,B 90.000,C 0.000} C_DIS
LIN {X 80.410,Y -41.634,Z -117.032,A -90.000,B 90.000,C 0.000} C_DIS
LIN {X 80.667,Y -41.576,Z -117.252,A -90.000,B 90.000,C 0.000} C_DIS
LIN {X 80.837,Y -41.548,Z -117.407,A -90.000,B 90.000,C 0.000} C_DIS
LIN {X 81.068,Y -41.504,Z -117.627,A -90.000,B 90.000,C 0.000} C_DIS
LIN {X 81.313,Y -41.457,Z -117.880,A -90.000,B 90.000,C 0.000} C_DIS
LIN {X 81.494,Y -41.405,Z -118.077,A -90.000,B 90.000,C 0.000} C_DIS
LIN {X 81.665,Y -41.356,Z -118.273,A -90.000,B 90.000,C 0.000} C_DIS
LIN {X 81.830,Y -41.308,Z -118.466,A -90.000,B 90.000,C 0.000} C_DIS
LIN {X 81.904,Y -41.291,Z -118.550,A -90.000,B 90.000,C 0.000} C_DIS
LIN {X 81.977,Y -41.270,Z -118.628,A -90.000,B 90.000,C 0.000} C_DIS
LIN {X 82.048,Y -41.250,Z -118.700,A -90.000,B 90.000,C 0.000} C_DIS
LIN {X 82.185,Y -41.210,Z -118.824,A -90.000,B 90.000,C 0.000} C_DIS
LIN {X 82.251,Y -41.191,Z -118.877,A -90.000,B 90.000,C 0.000} C_DIS
LIN {X 82.378,Y -41.155,Z -118.966,A -90.000,B 90.000,C 0.000} C_DIS
LIN {X 82.439,Y -41.137,Z -119.002,A -90.000,B 90.000,C 0.000} C_DIS
LIN {X 82.528,Y -41.112,Z -119.045,A -90.000,B 90.000,C 0.000} C_DIS
LIN {X 82.612,Y -41.088,Z -119.076,A -90.000,B 90.000,C 0.000} C_DIS
LIN {X 82.691,Y -41.065,Z -119.096,A -90.000,B 90.000,C 0.000} C_DIS
LIN {X 82.767,Y -41.044,Z -119.105,A -90.000,B 90.000,C 0.000} C_DIS
LIN {X 82.838,Y -41.023,Z -119.103,A -90.000,B 90.000,C 0.000} C_DIS
LIN {X 82.905,Y -41.004,Z -119.090,A -90.000,B 90.000,C 0.000} C_DIS
LIN {X 82.967,Y -40.987,Z -119.068,A -90.000,B 90.000,C 0.000} C_DIS
LIN {X 83.024,Y -40.970,Z -119.036,A -90.000,B 90.000,C 0.000} C_DIS
LIN {X 83.077,Y -40.955,Z -118.996,A -90.000,B 90.000,C 0.000} C_DIS
LIN {X 83.109,Y -40.947,Z -118.964,A -90.000,B 90.000,C 0.000} C_DIS
LIN {X 83.154,Y -40.935,Z -118.909,A -90.000,B 90.000,C 0.000} C_DIS
LIN {X 83.180,Y -40.929,Z -118.869,A -90.000,B 90.000,C 0.000} C_DIS
LIN {X 83.227,Y -40.917,Z -118.777,A -90.000,B 90.000,C 0.000} C_DIS
LIN {X 83.264,Y -40.909,Z -118.673,A -90.000,B 90.000,C 0.000} C_DIS
LIN {X 83.292,Y -40.903,Z -118.558,A -90.000,B 90.000,C 0.000} C_DIS
LIN {X 83.302,Y -40.902,Z -118.496,A -90.000,B 90.000,C 0.000} C_DIS
LIN {X 83.315,Y -40.901,Z -118.366,A -90.000,B 90.000,C 0.000} C_DIS
LIN {X 83.317,Y -40.902,Z -118.297,A -90.000,B 90.000,C 0.000} C_DIS
LIN {X 83.315,Y -40.907,Z -118.154,A -90.000,B 90.000,C 0.000} C_DIS
LIN {X 83.302,Y -40.915,Z -118.003,A -90.000,B 90.000,C 0.000} C_DIS
LIN {X 83.291,Y -40.920,Z -117.925,A -90.000,B 90.000,C 0.000} C_DIS
LIN {X 83.262,Y -40.933,Z -117.765,A -90.000,B 90.000,C 0.000} C_DIS
LIN {X 83.221,Y -40.950,Z -117.601,A -90.000,B 90.000,C 0.000} C_DIS
LIN {X 83.196,Y -40.960,Z -117.517,A -90.000,B 90.000,C 0.000} C_DIS
LIN {X 83.139,Y -40.982,Z -117.347,A -90.000,B 90.000,C 0.000} C_DIS
LIN {X 83.069,Y -41.009,Z -117.175,A -90.000,B 90.000,C 0.000} C_DIS
LIN {X 82.987,Y -41.039,Z -117.002,A -90.000,B 90.000,C 0.000} C_DIS
LIN {X 82.894,Y -41.073,Z -116.828,A -90.000,B 90.000,C 0.000} C_DIS
LIN {X 82.788,Y -41.112,Z -116.656,A -90.000,B 90.000,C 0.000} C_DIS
LIN {X 82.669,Y -41.154,Z -116.485,A -90.000,B 90.000,C 0.000} C_DIS
LIN {X 82.537,Y -41.204,Z -116.317,A -90.000,B 90.000,C 0.000} C_DIS
LIN {X 82.392,Y -41.257,Z -116.153,A -90.000,B 90.000,C 0.000} C_DIS
LIN {X 82.314,Y -41.285,Z -116.072,A -90.000,B 90.000,C 0.000} C_DIS
LIN {X 82.233,Y -41.308,Z -115.993,A -90.000,B 90.000,C 0.000} C_DIS
LIN {X 81.992,Y -41.393,Z -115.765,A -90.000,B 90.000,C 0.000} C_DIS
LIN {X 81.689,Y -41.498,Z -115.501,A -90.000,B 90.000,C 0.000} C_DIS
LIN {X 81.485,Y -41.568,Z -115.331,A -90.000,B 90.000,C 0.000} C_DIS
LIN {X 81.163,Y -41.642,Z -115.081,A -90.000,B 90.000,C 0.000} C_DIS
LIN {X 80.624,Y -41.768,Z -114.675,A -90.000,B 90.000,C 0.000} C_DIS
LIN {X 80.520,Y -41.792,Z -114.600,A -90.000,B 90.000,C 0.000} C_DIS
LIN {X 80.256,Y -41.853,Z -114.415,A -90.000,B 90.000,C 0.000} C_DIS
LIN {X 80.053,Y -41.899,Z -114.281,A -90.000,B 90.000,C 0.000} C_DIS
LIN {X 79.667,Y -41.984,Z -114.045,A -90.000,B 90.000,C 0.000} C_DIS
LIN {X 79.096,Y -42.113,Z -113.728,A -90.000,B 90.000,C 0.000} C_DIS
LIN {X 78.883,Y -42.161,Z -113.617,A -90.000,B 90.000,C 0.000} C_DIS
LIN {X 78.558,Y -42.232,Z -113.458,A -90.000,B 90.000,C 0.000} C_DIS
LIN {X 78.228,Y -42.301,Z -113.312,A -90.000,B 90.000,C 0.000} C_DIS
LIN {X 77.952,Y -42.355,Z -113.203,A -90.000,B 90.000,C 0.000} C_DIS
LIN {X 75.967,Y -42.560,Z -112.432,A -90.000,B 90.000,C 0.000} C_DIS
LIN {X 75.804,Y -42.576,Z -112.372,A -90.000,B 90.000,C 0.000} C_DIS
LIN {X 75.294,Y -42.628,Z -112.194,A -90.000,B 90.000,C 0.000} C_DIS
LIN {X 75.216,Y -42.635,Z -112.168,A -90.000,B 90.000,C 0.000} C_DIS
LIN {X 74.915,Y -42.664,Z -112.077,A -90.000,B 90.000,C 0.000} C_DIS
LIN {X 74.791,Y -42.673,Z -112.039,A -90.000,B 90.000,C 0.000} C_DIS
LIN {X 74.516,Y -42.691,Z -111.962,A -90.000,B 90.000,C 0.000} C_DIS
LIN {X 74.420,Y -42.693,Z -111.938,A -90.000,B 90.000,C 0.000} C_DIS
LIN {X 74.093,Y -42.691,Z -111.856,A -90.000,B 90.000,C 0.000} C_DIS
LIN {X 73.425,Y -42.683,Z -111.696,A -90.000,B 90.000,C 0.000} C_DIS
LIN {X 72.560,Y -42.671,Z -111.512,A -90.000,B 90.000,C 0.000} C_DIS
LIN {X 72.092,Y -42.664,Z -111.416,A -90.000,B 90.000,C 0.000} C_DIS
LIN {X 71.690,Y -42.658,Z -111.343,A -90.000,B 90.000,C 0.000} C_DIS
LIN {X 71.630,Y -42.657,Z -111.334,A -90.000,B 90.000,C 0.000} C_DIS
LIN {X 71.453,Y -42.652,Z -111.308,A -90.000,B 90.000,C 0.000} C_DIS
LIN {X 71.120,Y -42.625,Z -111.261,A -90.000,B 90.000,C 0.000} C_DIS
LIN {X 71.025,Y -42.617,Z -111.250,A -90.000,B 90.000,C 0.000} C_DIS
LIN {X 70.887,Y -42.603,Z -111.234,A -90.000,B 90.000,C 0.000} C_DIS
LIN {X 70.415,Y -42.527,Z -111.196,A -90.000,B 90.000,C 0.000} C_DIS
LIN {X 70.137,Y -42.482,Z -111.178,A -90.000,B 90.000,C 0.000} C_DIS
LIN {X 69.838,Y -42.436,Z -111.167,A -90.000,B 90.000,C 0.000} C_DIS
LIN {X 69.618,Y -42.402,Z -111.161,A -90.000,B 90.000,C 0.000} C_DIS
LIN {X 69.265,Y -42.348,Z -111.164,A -90.000,B 90.000,C 0.000} C_DIS
LIN {X 69.027,Y -42.312,Z -111.172,A -90.000,B 90.000,C 0.000} C_DIS
LIN {X 68.614,Y -42.250,Z -111.194,A -90.000,B 90.000,C 0.000} C_DIS
LIN {X 68.365,Y -42.213,Z -111.213,A -90.000,B 90.000,C 0.000} C_DIS
LIN {X 68.176,Y -42.181,Z -111.229,A -90.000,B 90.000,C 0.000} C_DIS
LIN {X 68.058,Y -42.160,Z -111.242,A -90.000,B 90.000,C 0.000} C_DIS
LIN {X 67.691,Y -42.096,Z -111.291,A -90.000,B 90.000,C 0.000} C_DIS
LIN {X 67.340,Y -42.008,Z -111.352,A -90.000,B 90.000,C 0.000} C_DIS
LIN {X 67.023,Y -41.930,Z -111.419,A -90.000,B 90.000,C 0.000} C_DIS
LIN {X 66.926,Y -41.904,Z -111.441,A -90.000,B 90.000,C 0.000} C_DIS
LIN {X 66.512,Y -41.794,Z -111.545,A -90.000,B 90.000,C 0.000} C_DIS
LIN {X 66.153,Y -41.700,Z -111.647,A -90.000,B 90.000,C 0.000} C_DIS
LIN {X 65.857,Y -41.624,Z -111.742,A -90.000,B 90.000,C 0.000} C_DIS
LIN {X 65.750,Y -41.598,Z -111.779,A -90.000,B 90.000,C 0.000} C_DIS
LIN {X 65.422,Y -41.514,Z -111.897,A -90.000,B 90.000,C 0.000} C_DIS
LIN {X 65.189,Y -41.456,Z -111.989,A -90.000,B 90.000,C 0.000} C_DIS
LIN {X 64.894,Y -41.384,Z -112.112,A -90.000,B 90.000,C 0.000} C_DIS
LIN {X 64.582,Y -41.308,Z -112.254,A -90.000,B 90.000,C 0.000} C_DIS
LIN {X 64.359,Y -41.255,Z -112.347,A -90.000,B 90.000,C 0.000} C_DIS
LIN {X 64.256,Y -41.229,Z -112.385,A -90.000,B 90.000,C 0.000} C_DIS
LIN {X 64.064,Y -41.177,Z -112.446,A -90.000,B 90.000,C 0.000} C_DIS
LIN {X 63.893,Y -41.126,Z -112.487,A -90.000,B 90.000,C 0.000} C_DIS
LIN {X 63.854,Y -41.115,Z -112.494,A -90.000,B 90.000,C 0.000} C_DIS
LIN {X 63.778,Y -41.091,Z -112.504,A -90.000,B 90.000,C 0.000} C_DIS
LIN {X 63.673,Y -41.058,Z -112.511,A -90.000,B 90.000,C 0.000} C_DIS
LIN {X 63.609,Y -41.037,Z -112.510,A -90.000,B 90.000,C 0.000} C_DIS
LIN {X 63.522,Y -41.006,Z -112.499,A -90.000,B 90.000,C 0.000} C_DIS
LIN {X 63.445,Y -40.977,Z -112.480,A -90.000,B 90.000,C 0.000} C_DIS
LIN {X 63.379,Y -40.949,Z -112.452,A -90.000,B 90.000,C 0.000} C_DIS
LIN {X 63.323,Y -40.924,Z -112.415,A -90.000,B 90.000,C 0.000} C_DIS
LIN {X 63.277,Y -40.900,Z -112.371,A -90.000,B 90.000,C 0.000} C_DIS
LIN {X 63.240,Y -40.878,Z -112.319,A -90.000,B 90.000,C 0.000} C_DIS
LIN {X 63.214,Y -40.858,Z -112.260,A -90.000,B 90.000,C 0.000} C_DIS
LIN {X 63.201,Y -40.845,Z -112.217,A -90.000,B 90.000,C 0.000} C_DIS
LIN {X 63.190,Y -40.829,Z -112.148,A -90.000,B 90.000,C 0.000} C_DIS
LIN {X 63.188,Y -40.819,Z -112.099,A -90.000,B 90.000,C 0.000} C_DIS
LIN {X 63.189,Y -40.810,Z -112.047,A -90.000,B 90.000,C 0.000} C_DIS
LIN {X 63.195,Y -40.802,Z -111.993,A -90.000,B 90.000,C 0.000} C_DIS
LIN {X 63.218,Y -40.788,Z -111.879,A -90.000,B 90.000,C 0.000} C_DIS
LIN {X 63.257,Y -40.779,Z -111.758,A -90.000,B 90.000,C 0.000} C_DIS
LIN {X 63.282,Y -40.776,Z -111.695,A -90.000,B 90.000,C 0.000} C_DIS
LIN {X 63.342,Y -40.773,Z -111.565,A -90.000,B 90.000,C 0.000} C_DIS
LIN {X 63.378,Y -40.773,Z -111.498,A -90.000,B 90.000,C 0.000} C_DIS
LIN {X 63.460,Y -40.776,Z -111.362,A -90.000,B 90.000,C 0.000} C_DIS
LIN {X 63.507,Y -40.779,Z -111.293,A -90.000,B 90.000,C 0.000} C_DIS
LIN {X 63.610,Y -40.789,Z -111.154,A -90.000,B 90.000,C 0.000} C_DIS
LIN {X 63.666,Y -40.796,Z -111.083,A -90.000,B 90.000,C 0.000} C_DIS
LIN {X 63.788,Y -40.813,Z -110.943,A -90.000,B 90.000,C 0.000} C_DIS
LIN {X 63.923,Y -40.835,Z -110.803,A -90.000,B 90.000,C 0.000} C_DIS
LIN {X 63.996,Y -40.848,Z -110.733,A -90.000,B 90.000,C 0.000} C_DIS
LIN {X 64.149,Y -40.877,Z -110.597,A -90.000,B 90.000,C 0.000} C_DIS
LIN {X 64.314,Y -40.912,Z -110.463,A -90.000,B 90.000,C 0.000} C_DIS
LIN {X 64.490,Y -40.952,Z -110.335,A -90.000,B 90.000,C 0.000} C_DIS
LIN {X 64.677,Y -40.997,Z -110.212,A -90.000,B 90.000,C 0.000} C_DIS
LIN {X 64.774,Y -41.022,Z -110.153,A -90.000,B 90.000,C 0.000} C_DIS
LIN {X 64.977,Y -41.075,Z -110.041,A -90.000,B 90.000,C 0.000} C_DIS
LIN {X 65.189,Y -41.135,Z -109.938,A -90.000,B 90.000,C 0.000} C_DIS
LIN {X 65.411,Y -41.200,Z -109.843,A -90.000,B 90.000,C 0.000} C_DIS
LIN {X 65.642,Y -41.275,Z -109.760,A -90.000,B 90.000,C 0.000} C_DIS
LIN {X 65.761,Y -41.308,Z -109.725,A -90.000,B 90.000,C 0.000} C_DIS
LIN {X 66.127,Y -41.426,Z -109.617,A -90.000,B 90.000,C 0.000} C_DIS
LIN {X 66.197,Y -41.449,Z -109.599,A -90.000,B 90.000,C 0.000} C_DIS
LIN {X 66.611,Y -41.556,Z -109.496,A -90.000,B 90.000,C 0.000} C_DIS
LIN {X 67.012,Y -41.661,Z -109.410,A -90.000,B 90.000,C 0.000} C_DIS
LIN {X 67.241,Y -41.721,Z -109.368,A -90.000,B 90.000,C 0.000} C_DIS
LIN {X 67.149,Y -41.686,Z -109.291,A -90.000,B 90.000,C 0.000} C_DIS
LIN {X 66.782,Y -41.544,Z -108.966,A -90.000,B 90.000,C 0.000} C_DIS
LIN {X 66.698,Y -41.509,Z -108.885,A -90.000,B 90.000,C 0.000} C_DIS
LIN {X 66.377,Y -41.332,Z -108.566,A -90.000,B 90.000,C 0.000} C_DIS
LIN {X 66.336,Y -41.308,Z -108.524,A -90.000,B 90.000,C 0.000} C_DIS
LIN {X 66.336,Y -60.000,Z -108.524,A -90.000,B 90.000,C 0.000} C_DIS
LIN {X 83.913,Y -60.000,Z -111.618,A -90.000,B 90.000,C 0.000} C_DIS
LIN {X 83.913,Y -41.308,Z -111.618,A -90.000,B 90.000,C 0.000} C_DIS
LIN {X 82.899,Y -41.562,Z -112.028,A -90.000,B 90.000,C 0.000} C_DIS
LIN {X 82.499,Y -41.663,Z -112.186,A -90.000,B 90.000,C 0.000} C_DIS
LIN {X 82.247,Y -41.721,Z -112.275,A -90.000,B 90.000,C 0.000} C_DIS
LIN {X 81.938,Y -41.789,Z -112.381,A -90.000,B 90.000,C 0.000} C_DIS
LIN {X 81.875,Y -41.800,Z -112.401,A -90.000,B 90.000,C 0.000} C_DIS
LIN {X 81.533,Y -41.846,Z -112.501,A -90.000,B 90.000,C 0.000} C_DIS
LIN {X 81.158,Y -41.897,Z -112.599,A -90.000,B 90.000,C 0.000} C_DIS
LIN {X 81.142,Y -41.899,Z -112.603,A -90.000,B 90.000,C 0.000} C_DIS
LIN {X 81.402,Y -41.838,Z -112.776,A -90.000,B 90.000,C 0.000} C_DIS
LIN {X 81.746,Y -41.755,Z -113.019,A -90.000,B 90.000,C 0.000} C_DIS
LIN {X 81.842,Y -41.730,Z -113.089,A -90.000,B 90.000,C 0.000} C_DIS
LIN {X 82.359,Y -41.540,Z -113.481,A -90.000,B 90.000,C 0.000} C_DIS
LIN {X 82.719,Y -41.403,Z -113.766,A -90.000,B 90.000,C 0.000} C_DIS
LIN {X 82.962,Y -41.308,Z -113.970,A -90.000,B 90.000,C 0.000} C_DIS
LIN {X 82.962,Y -60.000,Z -113.970,A -90.000,B 90.000,C 0.000} C_DIS
LIN {X -25.501,Y -60.000,Z -126.815,A -90.000,B 90.000,C 0.000} C_DIS
LIN {X -25.501,Y -41.308,Z -126.815,A -90.000,B 90.000,C 0.000} C_DIS
LIN {X -25.491,Y -41.338,Z -126.493,A -90.000,B 90.000,C 0.000} C_DIS
LIN {X -25.453,Y -41.415,Z -125.699,A -90.000,B 90.000,C 0.000} C_DIS
LIN {X -25.447,Y -41.455,Z -125.399,A -90.000,B 90.000,C 0.000} C_DIS
LIN {X -25.548,Y -41.484,Z -124.929,A -90.000,B 90.000,C 0.000} C_DIS
LIN {X -25.605,Y -41.505,Z -124.627,A -90.000,B 90.000,C 0.000} C_DIS
LIN {X -25.764,Y -41.548,Z -123.766,A -90.000,B 90.000,C 0.000} C_DIS
LIN {X -25.827,Y -41.554,Z -123.406,A -90.000,B 90.000,C 0.000} C_DIS
LIN {X -25.929,Y -41.580,Z -122.847,A -90.000,B 90.000,C 0.000} C_DIS
LIN {X -26.075,Y -41.601,Z -122.023,A -90.000,B 90.000,C 0.000} C_DIS
LIN {X -26.189,Y -41.597,Z -121.652,A -90.000,B 90.000,C 0.000} C_DIS
LIN {X -26.245,Y -41.595,Z -121.480,A -90.000,B 90.000,C 0.000} C_DIS
LIN {X -26.670,Y -41.632,Z -120.209,A -90.000,B 90.000,C 0.000} C_DIS
LIN {X -26.741,Y -41.633,Z -119.991,A -90.000,B 90.000,C 0.000} C_DIS
LIN {X -26.929,Y -41.627,Z -119.411,A -90.000,B 90.000,C 0.000} C_DIS
LIN {X -27.040,Y -41.636,Z -119.076,A -90.000,B 90.000,C 0.000} C_DIS
LIN {X -27.176,Y -41.648,Z -118.646,A -90.000,B 90.000,C 0.000} C_DIS
LIN {X -27.264,Y -41.650,Z -118.363,A -90.000,B 90.000,C 0.000} C_DIS
LIN {X -27.424,Y -41.641,Z -117.838,A -90.000,B 90.000,C 0.000} C_DIS
LIN {X -27.537,Y -41.634,Z -117.490,A -90.000,B 90.000,C 0.000} C_DIS
LIN {X -27.663,Y -41.642,Z -117.112,A -90.000,B 90.000,C 0.000} C_DIS
LIN {X -27.878,Y -41.651,Z -116.462,A -90.000,B 90.000,C 0.000} C_DIS
LIN {X -28.627,Y -41.650,Z -114.167,A -90.000,B 90.000,C 0.000} C_DIS
LIN {X -28.811,Y -41.649,Z -113.615,A -90.000,B 90.000,C 0.000} C_DIS
LIN {X -28.919,Y -41.642,Z -113.283,A -90.000,B 90.000,C 0.000} C_DIS
LIN {X -29.063,Y -41.616,Z -112.831,A -90.000,B 90.000,C 0.000} C_DIS
LIN {X -29.541,Y -41.512,Z -111.303,A -90.000,B 90.000,C 0.000} C_DIS
LIN {X -29.630,Y -41.499,Z -110.990,A -90.000,B 90.000,C 0.000} C_DIS
LIN {X -29.762,Y -41.481,Z -110.505,A -90.000,B 90.000,C 0.000} C_DIS
LIN {X -29.856,Y -41.471,Z -110.122,A -90.000,B 90.000,C 0.000} C_DIS
LIN {X -29.972,Y -41.456,Z -109.578,A -90.000,B 90.000,C 0.000} C_DIS
LIN {X -30.101,Y -41.434,Z -108.968,A -90.000,B 90.000,C 0.000} C_DIS
LIN {X -30.217,Y -41.411,Z -108.419,A -90.000,B 90.000,C 0.000} C_DIS
LIN {X -30.276,Y -41.383,Z -108.130,A -90.000,B 90.000,C 0.000} C_DIS
LIN {X -30.418,Y -41.308,Z -107.439,A -90.000,B 90.000,C 0.000} C_DIS
LIN {X -30.418,Y -60.000,Z -107.439,A -90.000,B 90.000,C 0.000} C_DIS
LIN {X -76.004,Y -60.000,Z -243.561,A -90.000,B 90.000,C 0.000} C_DIS
LIN {X -76.004,Y -42.069,Z -243.561,A -90.000,B 90.000,C 0.000} C_DIS
LIN {X -75.986,Y -42.018,Z -243.461,A -90.000,B 90.000,C 0.000} C_DIS
LIN {X -75.962,Y -41.964,Z -243.353,A -90.000,B 90.000,C 0.000} C_DIS
LIN {X -75.907,Y -41.868,Z -243.155,A -90.000,B 90.000,C 0.000} C_DIS
LIN {X -75.867,Y -41.804,Z -243.020,A -90.000,B 90.000,C 0.000} C_DIS
LIN {X -75.816,Y -41.741,Z -242.880,A -90.000,B 90.000,C 0.000} C_DIS
LIN {X -75.751,Y -41.671,Z -242.722,A -90.000,B 90.000,C 0.000} C_DIS
LIN {X -75.700,Y -41.621,Z -242.606,A -90.000,B 90.000,C 0.000} C_DIS
LIN {X -75.667,Y -41.593,Z -242.538,A -90.000,B 90.000,C 0.000} C_DIS
LIN {X -75.609,Y -41.549,Z -242.428,A -90.000,B 90.000,C 0.000} C_DIS
LIN {X -75.539,Y -41.499,Z -242.302,A -90.000,B 90.000,C 0.000} C_DIS
LIN {X -75.483,Y -41.465,Z -242.211,A -90.000,B 90.000,C 0.000} C_DIS
LIN {X -75.415,Y -41.429,Z -242.110,A -90.000,B 90.000,C 0.000} C_DIS
LIN {X -75.213,Y -41.334,Z -241.830,A -90.000,B 90.000,C 0.000} C_DIS
LIN {X -75.154,Y -41.308,Z -241.752,A -90.000,B 90.000,C 0.000} C_DIS
LIN {X -74.997,Y -41.243,Z -241.539,A -90.000,B 90.000,C 0.000} C_DIS
LIN {X -74.877,Y -41.192,Z -241.383,A -90.000,B 90.000,C 0.000} C_DIS
LIN {X -74.729,Y -41.134,Z -241.198,A -90.000,B 90.000,C 0.000} C_DIS
LIN {X -74.783,Y -41.162,Z -241.277,A -90.000,B 90.000,C 0.000} C_DIS
LIN {X -74.850,Y -41.191,Z -241.366,A -90.000,B 90.000,C 0.000} C_DIS
LIN {X -75.179,Y -41.326,Z -241.786,A -90.000,B 90.000,C 0.000} C_DIS
LIN {X -75.481,Y -41.441,Z -242.159,A -90.000,B 90.000,C 0.000} C_DIS
LIN {X -75.828,Y -41.566,Z -242.571,A -90.000,B 90.000,C 0.000} C_DIS
LIN {X -76.106,Y -41.658,Z -242.889,A -90.000,B 90.000,C 0.000} C_DIS
LIN {X -76.296,Y -41.716,Z -243.098,A -90.000,B 90.000,C 0.000} C_DIS
LIN {X -76.580,Y -41.797,Z -243.398,A -90.000,B 90.000,C 0.000} C_DIS
LIN {X -76.766,Y -41.843,Z -243.584,A -90.000,B 90.000,C 0.000} C_DIS
LIN {X -76.947,Y -41.882,Z -243.755,A -90.000,B 90.000,C 0.000} C_DIS
LIN {X -77.120,Y -41.913,Z -243.906,A -90.000,B 90.000,C 0.000} C_DIS
LIN {X -77.283,Y -41.934,Z -244.034,A -90.000,B 90.000,C 0.000} C_DIS
LIN {X -77.360,Y -41.940,Z -244.089,A -90.000,B 90.000,C 0.000} C_DIS
LIN {X -77.433,Y -41.944,Z -244.136,A -90.000,B 90.000,C 0.000} C_DIS
LIN {X -77.469,Y -41.945,Z -244.157,A -90.000,B 90.000,C 0.000} C_DIS
LIN {X -77.569,Y -41.941,Z -244.206,A -90.000,B 90.000,C 0.000} C_DIS
LIN {X -77.630,Y -41.935,Z -244.229,A -90.000,B 90.000,C 0.000} C_DIS
LIN {X -77.659,Y -41.930,Z -244.238,A -90.000,B 90.000,C 0.000} C_DIS
LIN {X -77.713,Y -41.918,Z -244.248,A -90.000,B 90.000,C 0.000} C_DIS
LIN {X -77.762,Y -41.902,Z -244.248,A -90.000,B 90.000,C 0.000} C_DIS
LIN {X -77.806,Y -41.883,Z -244.238,A -90.000,B 90.000,C 0.000} C_DIS
LIN {X -77.826,Y -41.872,Z -244.230,A -90.000,B 90.000,C 0.000} C_DIS
LIN {X -77.862,Y -41.846,Z -244.206,A -90.000,B 90.000,C 0.000} C_DIS
LIN {X -77.896,Y -41.812,Z -244.167,A -90.000,B 90.000,C 0.000} C_DIS
LIN {X -77.909,Y -41.795,Z -244.145,A -90.000,B 90.000,C 0.000} C_DIS
LIN {X -77.921,Y -41.777,Z -244.120,A -90.000,B 90.000,C 0.000} C_DIS
LIN {X -77.928,Y -41.758,Z -244.092,A -90.000,B 90.000,C 0.000} C_DIS
LIN {X -77.942,Y -41.715,Z -244.026,A -90.000,B 90.000,C 0.000} C_DIS
LIN {X -77.948,Y -41.666,Z -243.947,A -90.000,B 90.000,C 0.000} C_DIS
LIN {X -77.948,Y -41.640,Z -243.902,A -90.000,B 90.000,C 0.000} C_DIS
LIN {X -77.943,Y -41.583,Z -243.802,A -90.000,B 90.000,C 0.000} C_DIS
LIN {X -77.920,Y -41.488,Z -243.627,A -90.000,B 90.000,C 0.000} C_DIS
LIN {X -77.905,Y -41.447,Z -243.561,A -90.000,B 90.000,C 0.000} C_DIS
LIN {X -77.882,Y -41.381,Z -243.435,A -90.000,B 90.000,C 0.000} C_DIS
LIN {X -77.851,Y -41.308,Z -243.292,A -90.000,B 90.000,C 0.000} C_DIS
LIN {X -77.847,Y -41.305,Z -243.271,A -90.000,B 90.000,C 0.000} C_DIS
LIN {X -77.843,Y -41.286,Z -243.235,A -90.000,B 90.000,C 0.000} C_DIS
LIN {X -77.846,Y -41.269,Z -243.208,A -90.000,B 90.000,C 0.000} C_DIS
LIN {X -77.860,Y -41.248,Z -243.180,A -90.000,B 90.000,C 0.000} C_DIS
LIN {X -77.885,Y -41.232,Z -243.167,A -90.000,B 90.000,C 0.000} C_DIS
LIN {X -77.918,Y -41.220,Z -243.167,A -90.000,B 90.000,C 0.000} C_DIS
LIN {X -77.945,Y -41.215,Z -243.174,A -90.000,B 90.000,C 0.000} C_DIS
LIN {X -77.974,Y -41.212,Z -243.186,A -90.000,B 90.000,C 0.000} C_DIS
LIN {X -78.039,Y -41.210,Z -243.220,A -90.000,B 90.000,C 0.000} C_DIS
LIN {X -78.146,Y -41.217,Z -243.294,A -90.000,B 90.000,C 0.000} C_DIS
LIN {X -78.252,Y -41.233,Z -243.382,A -90.000,B 90.000,C 0.000} C_DIS
LIN {X -78.343,Y -41.253,Z -243.471,A -90.000,B 90.000,C 0.000} C_DIS
LIN {X -78.409,Y -41.275,Z -243.547,A -90.000,B 90.000,C 0.000} C_DIS
LIN {X -78.422,Y -41.283,Z -243.567,A -90.000,B 90.000,C 0.000} C_DIS
LIN {X -78.433,Y -41.293,Z -243.591,A -90.000,B 90.000,C 0.000} C_DIS
LIN {X -78.431,Y -41.301,Z -243.605,A -90.000,B 90.000,C 0.000} C_DIS
LIN {X -78.422,Y -41.306,Z -243.608,A -90.000,B 90.000,C 0.000} C_DIS
LIN {X -78.406,Y -41.311,Z -243.606,A -90.000,B 90.000,C 0.000} C_DIS
LIN {X -78.383,Y -41.314,Z -243.598,A -90.000,B 90.000,C 0.000} C_DIS
LIN {X -78.353,Y -41.316,Z -243.583,A -90.000,B 90.000,C 0.000} C_DIS
LIN {X -78.313,Y -41.308,Z -243.561,A -90.000,B 90.000,C 0.000} C_DIS
LIN {X -76.699,Y -41.308,Z -242.621,A -90.000,B 90.000,C 0.000} C_DIS
LIN {X -70.921,Y -41.308,Z -239.371,A -90.000,B 90.000,C 0.000} C_DIS
LIN {X -70.376,Y -41.308,Z -239.077,A -90.000,B 90.000,C 0.000} C_DIS
LIN {X -62.171,Y -41.308,Z -234.728,A -90.000,B 90.000,C 0.000} C_DIS
LIN {X -58.363,Y -41.308,Z -232.790,A -90.000,B 90.000,C 0.000} C_DIS
LIN {X -53.644,Y -41.308,Z -230.431,A -90.000,B 90.000,C 0.000} C_DIS
LIN {X -52.575,Y -41.308,Z -229.902,A -90.000,B 90.000,C 0.000} C_DIS
LIN {X -50.401,Y -41.308,Z -228.843,A -90.000,B 90.000,C 0.000} C_DIS
LIN {X -46.947,Y -41.308,Z -227.187,A -90.000,B 90.000,C 0.000} C_DIS
LIN {X -45.243,Y -41.308,Z -226.396,A -90.000,B 90.000,C 0.000} C_DIS
LIN {X -41.599,Y -41.308,Z -224.674,A -90.000,B 90.000,C 0.000} C_DIS
LIN {X -37.247,Y -41.308,Z -222.680,A -90.000,B 90.000,C 0.000} C_DIS
LIN {X -36.527,Y -41.308,Z -222.337,A -90.000,B 90.000,C 0.000} C_DIS
LIN {X -35.174,Y -41.308,Z -221.704,A -90.000,B 90.000,C 0.000} C_DIS
LIN {X -33.159,Y -41.308,Z -220.790,A -90.000,B 90.000,C 0.000} C_DIS
LIN {X -31.326,Y -41.308,Z -219.981,A -90.000,B 90.000,C 0.000} C_DIS
LIN {X -30.240,Y -41.308,Z -219.517,A -90.000,B 90.000,C 0.000} C_DIS
LIN {X -27.083,Y -41.308,Z -218.038,A -90.000,B 90.000,C 0.000} C_DIS
LIN {X -23.944,Y -41.308,Z -216.558,A -90.000,B 90.000,C 0.000} C_DIS
LIN {X -23.074,Y -41.308,Z -216.113,A -90.000,B 90.000,C 0.000} C_DIS
LIN {X -21.089,Y -41.308,Z -215.064,A -90.000,B 90.000,C 0.000} C_DIS
LIN {X -19.174,Y -41.308,Z -214.141,A -90.000,B 90.000,C 0.000} C_DIS
LIN {X -18.798,Y -41.308,Z -213.964,A -90.000,B 90.000,C 0.000} C_DIS
LIN {X -15.714,Y -41.308,Z -212.317,A -90.000,B 90.000,C 0.000} C_DIS
LIN {X -14.086,Y -41.308,Z -211.402,A -90.000,B 90.000,C 0.000} C_DIS
LIN {X -12.446,Y -41.308,Z -210.415,A -90.000,B 90.000,C 0.000} C_DIS
LIN {X -9.775,Y -41.308,Z -208.729,A -90.000,B 90.000,C 0.000} C_DIS
LIN {X -7.693,Y -41.308,Z -207.330,A -90.000,B 90.000,C 0.000} C_DIS
LIN {X -5.600,Y -41.308,Z -206.061,A -90.000,B 90.000,C 0.000} C_DIS
LIN {X -4.299,Y -41.308,Z -205.134,A -90.000,B 90.000,C 0.000} C_DIS
LIN {X -1.671,Y -41.308,Z -203.336,A -90.000,B 90.000,C 0.000} C_DIS
LIN {X 1.046,Y -41.308,Z -201.104,A -90.000,B 90.000,C 0.000} C_DIS
LIN {X 1.982,Y -41.308,Z -200.376,A -90.000,B 90.000,C 0.000} C_DIS
LIN {X 5.265,Y -41.308,Z -197.252,A -90.000,B 90.000,C 0.000} C_DIS
LIN {X 5.482,Y -41.308,Z -197.059,A -90.000,B 90.000,C 0.000} C_DIS
LIN {X 5.598,Y -41.308,Z -196.943,A -90.000,B 90.000,C 0.000} C_DIS
LIN {X 8.562,Y -41.308,Z -193.684,A -90.000,B 90.000,C 0.000} C_DIS
LIN {X 8.693,Y -41.308,Z -193.543,A -90.000,B 90.000,C 0.000} C_DIS
LIN {X 11.673,Y -41.308,Z -190.051,A -90.000,B 90.000,C 0.000} C_DIS
LIN {X 14.548,Y -41.308,Z -186.630,A -90.000,B 90.000,C 0.000} C_DIS
LIN {X 14.601,Y -41.308,Z -186.563,A -90.000,B 90.000,C 0.000} C_DIS
LIN {X 17.224,Y -41.308,Z -183.565,A -90.000,B 90.000,C 0.000} C_DIS
LIN {X 17.303,Y -41.308,Z -183.468,A -90.000,B 90.000,C 0.000} C_DIS
LIN {X 17.506,Y -41.308,Z -183.235,A -90.000,B 90.000,C 0.000} C_DIS
LIN {X 17.587,Y -41.308,Z -183.147,A -90.000,B 90.000,C 0.000} C_DIS
LIN {X 19.984,Y -41.308,Z -180.680,A -90.000,B 90.000,C 0.000} C_DIS
LIN {X 20.245,Y -41.308,Z -180.417,A -90.000,B 90.000,C 0.000} C_DIS
LIN {X 22.284,Y -41.308,Z -178.458,A -90.000,B 90.000,C 0.000} C_DIS
LIN {X 23.317,Y -41.308,Z -177.450,A -90.000,B 90.000,C 0.000} C_DIS
LIN {X 23.817,Y -41.308,Z -176.964,A -90.000,B 90.000,C 0.000} C_DIS
LIN {X 24.353,Y -41.308,Z -176.459,A -90.000,B 90.000,C 0.000} C_DIS
LIN {X 25.984,Y -41.308,Z -174.797,A -90.000,B 90.000,C 0.000} C_DIS
LIN {X 26.063,Y -41.308,Z -174.719,A -90.000,B 90.000,C 0.000} C_DIS
LIN {X 26.517,Y -41.308,Z -174.197,A -90.000,B 90.000,C 0.000} C_DIS
LIN {X 27.680,Y -41.308,Z -172.849,A -90.000,B 90.000,C 0.000} C_DIS
LIN {X 27.888,Y -41.308,Z -172.573,A -90.000,B 90.000,C 0.000} C_DIS
LIN {X 28.053,Y -41.308,Z -172.357,A -90.000,B 90.000,C 0.000} C_DIS
LIN {X 29.042,Y -41.308,Z -171.082,A -90.000,B 90.000,C 0.000} C_DIS
LIN {X 29.701,Y -41.308,Z -170.121,A -90.000,B 90.000,C 0.000} C_DIS
LIN {X 30.450,Y -41.308,Z -169.064,A -90.000,B 90.000,C 0.000} C_DIS
LIN {X 31.367,Y -41.308,Z -167.629,A -90.000,B 90.000,C 0.000} C_DIS
LIN {X 31.759,Y -41.308,Z -167.035,A -90.000,B 90.000,C 0.000} C_DIS
LIN {X 31.795,Y -41.308,Z -166.980,A -90.000,B 90.000,C 0.000} C_DIS
LIN {X 32.016,Y -41.308,Z -166.602,A -90.000,B 90.000,C 0.000} C_DIS
LIN {X 33.226,Y -41.308,Z -164.588,A -90.000,B 90.000,C 0.000} C_DIS
LIN {X 33.816,Y -41.308,Z -163.527,A -90.000,B 90.000,C 0.000} C_DIS
LIN {X 34.651,Y -41.308,Z -162.055,A -90.000,B 90.000,C 0.000} C_DIS
LIN {X 35.704,Y -41.308,Z -160.041,A -90.000,B 90.000,C 0.000} C_DIS
LIN {X 36.026,Y -41.308,Z -159.431,A -90.000,B 90.000,C 0.000} C_DIS
LIN {X 37.228,Y -41.308,Z -156.954,A -90.000,B 90.000,C 0.000} C_DIS
LIN {X 37.840,Y -41.308,Z -155.569,A -90.000,B 90.000,C 0.000} C_DIS
LIN {X 38.386,Y -41.308,Z -154.400,A -90.000,B 90.000,C 0.000} C_DIS
LIN {X 38.932,Y -41.308,Z -153.055,A -90.000,B 90.000,C 0.000} C_DIS
LIN {X 39.476,Y -41.308,Z -151.859,A -90.000,B 90.000,C 0.000} C_DIS
LIN {X 39.754,Y -41.308,Z -151.136,A -90.000,B 90.000,C 0.000} C_DIS
LIN {X 40.468,Y -41.308,Z -149.587,A -90.000,B 90.000,C 0.000} C_DIS
LIN {X 40.660,Y -41.308,Z -149.160,A -90.000,B 90.000,C 0.000} C_DIS
LIN {X 40.690,Y -41.308,Z -149.103,A -90.000,B 90.000,C 0.000} C_DIS
LIN {X 40.783,Y -41.308,Z -148.884,A -90.000,B 90.000,C 0.000} C_DIS
LIN {X 41.087,Y -41.308,Z -148.270,A -90.000,B 90.000,C 0.000} C_DIS
LIN {X 41.586,Y -41.308,Z -147.200,A -90.000,B 90.000,C 0.000} C_DIS
LIN {X 41.716,Y -41.308,Z -146.934,A -90.000,B 90.000,C 0.000} C_DIS
LIN {X 42.132,Y -41.308,Z -146.197,A -90.000,B 90.000,C 0.000} C_DIS
LIN {X 42.761,Y -41.308,Z -144.956,A -90.000,B 90.000,C 0.000} C_DIS
LIN {X 42.930,Y -41.308,Z -144.685,A -90.000,B 90.000,C 0.000} C_DIS
LIN {X 43.920,Y -41.308,Z -143.161,A -90.000,B 90.000,C 0.000} C_DIS
LIN {X 44.094,Y -41.308,Z -142.880,A -90.000,B 90.000,C 0.000} C_DIS
LIN {X 44.245,Y -41.308,Z -142.639,A -90.000,B 90.000,C 0.000} C_DIS
LIN {X 44.579,Y -41.308,Z -142.179,A -90.000,B 90.000,C 0.000} C_DIS
LIN {X 45.592,Y -41.308,Z -140.694,A -90.000,B 90.000,C 0.000} C_DIS
LIN {X 46.733,Y -41.308,Z -139.290,A -90.000,B 90.000,C 0.000} C_DIS
LIN {X 47.229,Y -41.308,Z -138.661,A -90.000,B 90.000,C 0.000} C_DIS
LIN {X 47.438,Y -41.308,Z -138.421,A -90.000,B 90.000,C 0.000} C_DIS
LIN {X 48.015,Y -41.308,Z -137.767,A -90.000,B 90.000,C 0.000} C_DIS
LIN {X 48.923,Y -41.308,Z -136.680,A -90.000,B 90.000,C 0.000} C_DIS
LIN {X 49.133,Y -41.308,Z -136.439,A -90.000,B 90.000,C 0.000} C_DIS
LIN {X 50.197,Y -41.308,Z -135.270,A -90.000,B 90.000,C 0.000} C_DIS
LIN {X 50.987,Y -41.308,Z -134.408,A -90.000,B 90.000,C 0.000} C_DIS
LIN {X 51.727,Y -41.308,Z -133.644,A -90.000,B 90.000,C 0.000} C_DIS
LIN {X 52.989,Y -41.308,Z -132.170,A -90.000,B 90.000,C 0.000} C_DIS
LIN {X 54.747,Y -41.308,Z -130.113,A -90.000,B 90.000,C 0.000} C_DIS
LIN {X 56.350,Y -41.308,Z -127.563,A -90.000,B 90.000,C 0.000} C_DIS
LIN {X 56.816,Y -41.308,Z -126.800,A -90.000,B 90.000,C 0.000} C_DIS
LIN {X 57.778,Y -41.308,Z -125.111,A -90.000,B 90.000,C 0.000} C_DIS
LIN {X 58.977,Y -41.308,Z -122.826,A -90.000,B 90.000,C 0.000} C_DIS
LIN {X 59.052,Y -41.308,Z -122.710,A -90.000,B 90.000,C 0.000} C_DIS
LIN {X 59.137,Y -41.308,Z -122.542,A -90.000,B 90.000,C 0.000} C_DIS
LIN {X 61.305,Y -41.308,Z -118.681,A -90.000,B 90.000,C 0.000} C_DIS
LIN {X 61.816,Y -41.308,Z -117.681,A -90.000,B 90.000,C 0.000} C_DIS
LIN {X 63.316,Y -41.308,Z -114.863,A -90.000,B 90.000,C 0.000} C_DIS
LIN {X 63.941,Y -41.308,Z -113.660,A -90.000,B 90.000,C 0.000} C_DIS
LIN {X 64.986,Y -41.308,Z -111.369,A -90.000,B 90.000,C 0.000} C_DIS
LIN {X 65.035,Y -41.308,Z -111.252,A -90.000,B 90.000,C 0.000} C_DIS
LIN {X 66.178,Y -41.308,Z -108.849,A -90.000,B 90.000,C 0.000} C_DIS
LIN {X 66.370,Y -41.308,Z -108.456,A -90.000,B 90.000,C 0.000} C_DIS
LIN {X 66.457,Y -41.308,Z -108.259,A -90.000,B 90.000,C 0.000} C_DIS
LIN {X 66.929,Y -41.308,Z -107.161,A -90.000,B 90.000,C 0.000} C_DIS
LIN {X 67.618,Y -41.308,Z -105.261,A -90.000,B 90.000,C 0.000} C_DIS
LIN {X 67.856,Y -41.308,Z -104.317,A -90.000,B 90.000,C 0.000} C_DIS
LIN {X 68.063,Y -41.308,Z -103.614,A -90.000,B 90.000,C 0.000} C_DIS
LIN {X 68.100,Y -41.308,Z -103.401,A -90.000,B 90.000,C 0.000} C_DIS
LIN {X 68.250,Y -41.308,Z -102.360,A -90.000,B 90.000,C 0.000} C_DIS
LIN {X 68.219,Y -41.308,Z -101.266,A -90.000,B 90.000,C 0.000} C_DIS
LIN {X 68.192,Y -41.308,Z -101.151,A -90.000,B 90.000,C 0.000} C_DIS
LIN {X 67.579,Y -41.308,Z -99.316,A -90.000,B 90.000,C 0.000} C_DIS
LIN {X 67.482,Y -41.308,Z -99.107,A -90.000,B 90.000,C 0.000} C_DIS
LIN {X 67.365,Y -41.308,Z -98.892,A -90.000,B 90.000,C 0.000} C_DIS
LIN {X 66.405,Y -41.308,Z -97.093,A -90.000,B 90.000,C 0.000} C_DIS
LIN {X 65.718,Y -41.308,Z -95.681,A -90.000,B 90.000,C 0.000} C_DIS
LIN {X 65.411,Y -41.308,Z -94.979,A -90.000,B 90.000,C 0.000} C_DIS
LIN {X 65.324,Y -41.308,Z -94.711,A -90.000,B 90.000,C 0.000} C_DIS
LIN {X 64.889,Y -41.308,Z -92.960,A -90.000,B 90.000,C 0.000} C_DIS
LIN {X 64.642,Y -41.308,Z -92.023,A -90.000,B 90.000,C 0.000} C_DIS
LIN {X 64.603,Y -41.308,Z -91.743,A -90.000,B 90.000,C 0.000} C_DIS
LIN {X 64.583,Y -41.308,Z -91.564,A -90.000,B 90.000,C 0.000} C_DIS
LIN {X 64.583,Y -41.308,Z -91.397,A -90.000,B 90.000,C 0.000} C_DIS
LIN {X 64.553,Y -41.308,Z -87.997,A -90.000,B 90.000,C 0.000} C_DIS
LIN {X 64.556,Y -41.308,Z -87.920,A -90.000,B 90.000,C 0.000} C_DIS
LIN {X 64.556,Y -41.308,Z -87.866,A -90.000,B 90.000,C 0.000} C_DIS
LIN {X 64.567,Y -41.308,Z -87.597,A -90.000,B 90.000,C 0.000} C_DIS
LIN {X 64.641,Y -41.308,Z -86.084,A -90.000,B 90.000,C 0.000} C_DIS
LIN {X 64.610,Y -41.308,Z -84.536,A -90.000,B 90.000,C 0.000} C_DIS
LIN {X 64.621,Y -41.308,Z -84.254,A -90.000,B 90.000,C 0.000} C_DIS
LIN {X 64.647,Y -41.308,Z -84.042,A -90.000,B 90.000,C 0.000} C_DIS
LIN {X 64.649,Y -41.308,Z -83.811,A -90.000,B 90.000,C 0.000} C_DIS
LIN {X 64.652,Y -41.308,Z -82.505,A -90.000,B 90.000,C 0.000} C_DIS
LIN {X 64.561,Y -41.308,Z -80.961,A -90.000,B 90.000,C 0.000} C_DIS
LIN {X 64.557,Y -41.308,Z -80.797,A -90.000,B 90.000,C 0.000} C_DIS
LIN {X 64.531,Y -41.308,Z -80.684,A -90.000,B 90.000,C 0.000} C_DIS
LIN {X 64.353,Y -41.308,Z -80.016,A -90.000,B 90.000,C 0.000} C_DIS
LIN {X 64.324,Y -41.308,Z -79.788,A -90.000,B 90.000,C 0.000} C_DIS
LIN {X 64.265,Y -41.308,Z -79.061,A -90.000,B 90.000,C 0.000} C_DIS
LIN {X 64.258,Y -41.308,Z -78.929,A -90.000,B 90.000,C 0.000} C_DIS
LIN {X 64.313,Y -41.308,Z -78.555,A -90.000,B 90.000,C 0.000} C_DIS
LIN {X 64.352,Y -41.308,Z -78.380,A -90.000,B 90.000,C 0.000} C_DIS
LIN {X 64.608,Y -41.308,Z -77.881,A -90.000,B 90.000,C 0.000} C_DIS
LIN {X 63.524,Y -41.308,Z -75.967,A -90.000,B 90.000,C 0.000} C_DIS
LIN {X 63.490,Y -41.308,Z -75.895,A -90.000,B 90.000,C 0.000} C_DIS
LIN {X 63.343,Y -41.308,Z -75.563,A -90.000,B 90.000,C 0.000} C_DIS
LIN {X 61.746,Y -41.308,Z -75.486,A -90.000,B 90.000,C 0.000} C_DIS
LIN {X 61.348,Y -41.308,Z -75.438,A -90.000,B 90.000,C 0.000} C_DIS
LIN {X 60.840,Y -41.308,Z -75.260,A -90.000,B 90.000,C 0.000} C_DIS
LIN {X 60.084,Y -41.308,Z -75.479,A -90.000,B 90.000,C 0.000} C_DIS
LIN {X 59.914,Y -41.308,Z -75.506,A -90.000,B 90.000,C 0.000} C_DIS
LIN {X 59.049,Y -41.308,Z -75.609,A -90.000,B 90.000,C 0.000} C_DIS
LIN {X 58.117,Y -41.308,Z -75.621,A -90.000,B 90.000,C 0.000} C_DIS
LIN {X 56.497,Y -41.308,Z -75.978,A -90.000,B 90.000,C 0.000} C_DIS
LIN {X 55.339,Y -41.308,Z -76.204,A -90.000,B 90.000,C 0.000} C_DIS
LIN {X 54.352,Y -41.308,Z -76.559,A -90.000,B 90.000,C 0.000} C_DIS
LIN {X 54.184,Y -41.308,Z -76.618,A -90.000,B 90.000,C 0.000} C_DIS
LIN {X 51.662,Y -41.308,Z -77.455,A -90.000,B 90.000,C 0.000} C_DIS
LIN {X 50.843,Y -41.308,Z -77.708,A -90.000,B 90.000,C 0.000} C_DIS
LIN {X 48.217,Y -41.308,Z -78.762,A -90.000,B 90.000,C 0.000} C_DIS
LIN {X 48.210,Y -41.308,Z -78.765,A -90.000,B 90.000,C 0.000} C_DIS
LIN {X 48.093,Y -41.308,Z -78.858,A -90.000,B 90.000,C 0.000} C_DIS
LIN {X 47.963,Y -41.308,Z -79.183,A -90.000,B 90.000,C 0.000} C_DIS
LIN {X 47.865,Y -41.308,Z -79.333,A -90.000,B 90.000,C 0.000} C_DIS
LIN {X 47.215,Y -41.308,Z -80.179,A -90.000,B 90.000,C 0.000} C_DIS
LIN {X 47.383,Y -41.308,Z -80.988,A -90.000,B 90.000,C 0.000} C_DIS
LIN {X 48.144,Y -41.308,Z -81.965,A -90.000,B 90.000,C 0.000} C_DIS
LIN {X 48.217,Y -41.308,Z -82.129,A -90.000,B 90.000,C 0.000} C_DIS
LIN {X 48.241,Y -41.308,Z -82.306,A -90.000,B 90.000,C 0.000} C_DIS
LIN {X 48.281,Y -41.308,Z -83.066,A -90.000,B 90.000,C 0.000} C_DIS
LIN {X 48.824,Y -41.308,Z -83.710,A -90.000,B 90.000,C 0.000} C_DIS
LIN {X 49.699,Y -41.308,Z -85.390,A -90.000,B 90.000,C 0.000} C_DIS
LIN {X 49.886,Y -41.308,Z -85.631,A -90.000,B 90.000,C 0.000} C_DIS
LIN {X 50.840,Y -41.308,Z -86.945,A -90.000,B 90.000,C 0.000} C_DIS
LIN {X 51.686,Y -41.308,Z -88.413,A -90.000,B 90.000,C 0.000} C_DIS
LIN {X 51.932,Y -41.308,Z -88.710,A -90.000,B 90.000,C 0.000} C_DIS
LIN {X 53.109,Y -41.308,Z -90.547,A -90.000,B 90.000,C 0.000} C_DIS
LIN {X 53.229,Y -41.308,Z -90.756,A -90.000,B 90.000,C 0.000} C_DIS
LIN {X 54.128,Y -41.308,Z -92.725,A -90.000,B 90.000,C 0.000} C_DIS
LIN {X 54.168,Y -41.308,Z -92.800,A -90.000,B 90.000,C 0.000} C_DIS
LIN {X 54.274,Y -41.308,Z -93.129,A -90.000,B 90.000,C 0.000} C_DIS
LIN {X 55.524,Y -41.308,Z -97.374,A -90.000,B 90.000,C 0.000} C_DIS
LIN {X 55.546,Y -41.308,Z -97.522,A -90.000,B 90.000,C 0.000} C_DIS
LIN {X 55.571,Y -41.308,Z -97.758,A -90.000,B 90.000,C 0.000} C_DIS
LIN {X 55.570,Y -41.308,Z -97.807,A -90.000,B 90.000,C 0.000} C_DIS
LIN {X 55.656,Y -41.308,Z -98.754,A -90.000,B 90.000,C 0.000} C_DIS
LIN {X 55.776,Y -41.308,Z -101.506,A -90.000,B 90.000,C 0.000} C_DIS
LIN {X 55.777,Y -41.308,Z -101.529,A -90.000,B 90.000,C 0.000} C_DIS
LIN {X 55.772,Y -41.308,Z -101.655,A -90.000,B 90.000,C 0.000} C_DIS
LIN {X 55.518,Y -41.308,Z -104.242,A -90.000,B 90.000,C 0.000} C_DIS
